METHOD PRIVATE REAL_TO_WHOLE_AND_FRACTION : BOOL
VAR_INPUT
	nReal		:	REAL;				// The real number you want to split into whole and fractional parts
END_VAR
VAR_OUTPUT
	nWhole		:	INT;				// The whole part of the input
	nFraction	:	UINT;				// The fractional part of the input (multiplied by 1000)
END_VAR
VAR
	sTemp		: STRING;
END_VAR
sTemp := REAL_TO_STRING(nReal);
nWhole := STRING_TO_INT(LEFT(sTEMP, FIND(sTemp, '.')));
sTemp := DELETE(sTEmp, FIND(sTemp, '.'), 1);
CASE LEN(sTemp) OF
	0:		sTemp := '000';
	1:		sTemp := CONCAT(sTemp, '00');
	2:		sTemp := CONCAT(sTemp, '0');
	ELSE	sTemp := LEFT(sTemp, 3);
END_CASE
nFraction := STRING_TO_UINT(sTemp);
REAL_TO_WHOLE_AND_FRACTION := TRUE;
END_METHOD

METHOD PRIVATE WHOLE_AND_FRACTION_TO_REAL : BOOL
VAR_INPUT
	nWhole		: INT;					// The whole part of the numbers you want to combine into real
	nFraction	: UINT;					// The fractional part of the numbers you want to combine into real
END_VAR
VAR_OUTPUT
	nReal 		: REAL;					// The result real number
END_VAR
VAR
	sTemp		: STRING;
END_VAR
nReal := STRING_TO_REAL(CONCAT(CONCAT(INT_TO_STRING(nWhole),'.'), UINT_TO_STRING(nFraction)));
WHOLE_AND_FRACTION_TO_REAL := TRUE;
END_METHOD

END_FUNCTION_BLOCK

// ---- POUs/CNC_1/CNC_1.TcPOU
PROGRAM CNC_1
VAR	(* Control *)
	nState						: UDINT;
	nStatePrevious				: UDINT;
	sState						: STRING(500);
	fbCycleTime					: TON;
	nCycleTime					: REAL;
	bError						: BOOL;
END_VAR
VAR (* LastStates *)
	anLastStates				: ARRAY[0..500] OF UDINT;
    iLastStates					: INT;
END_VAR
VAR (* Var IO *)
	{attribute 'TcLinkTo' := '		.fbMoveUpper.i_bBasePos	:= TIIB(13)^Channel 2^Input;
									.fbMoveUpper.i_bWorkPos	:= TIIB(13)^Channel 1^Input;
									.fbMoveUpper.q_bBasePos	:= TIIB(14)^Channel 2^Output;
									.fbMoveUpper.q_bWorkPos	:= TIIB(14)^Channel 1^Output;
									.fbMoveLower.i_bBasePos	:= TIIB(13)^Channel 4^Input;
									.fbMoveLower.i_bWorkPos	:= TIIB(13)^Channel 3^Input;
									.fbMoveLower.q_bBasePos	:= TIIB(14)^Channel 4^Output;
									.fbMoveLower.q_bWorkPos	:= TIIB(14)^Channel 3^Output;
									.fbLock.i_bBasePos	:= TIIB(13)^Channel 5^Input;
									.fbLock.i_bWorkPos	:= TIIB(13)^Channel 6^Input;
									.fbLock.q_bWorkPos	:= TIIB(14)^Channel 5^Output;
									.q_bToolCheckBlower := TIIB(14)^Channel 6^Output;
									.fbVisePos.arrRaw[0]	:= TIIB(10)^Module 1 (IOL_I_4byte)^TxPDO^input byte 0;	
									.fbVisePos.arrRaw[1] 	:= TIIB(10)^Module 1 (IOL_I_4byte)^TxPDO^input byte 1;
									.fbVisePos.arrRaw[2]	:= TIIB(10)^Module 1 (IOL_I_4byte)^TxPDO^input byte 2;
									.fbVisePos.arrRaw[3]	:= TIIB(10)^Module 1 (IOL_I_4byte)^TxPDO^input byte 3;
									.fbVisePos.nState		:= TIIB(10)^IO-Link DeviceState Inputs^Status of IO-Link Port 1;'}
	fbCncServoVise				: FB_CNC_Servo;	

END_VAR
VAR (* OPC_UA *)
	stCNC_Data					: POINTER TO OPC_CNC_Data_Collection;
	tHeartBeatDelay				: TON;
	bCNCHandshakeTimeout		:	BOOL;
	tCNCHandshakeTimer			:	TON;
	bCNCMidwareShutdownPossible	: 	BOOL;	//20, 40, 11400, 
	bShutdownIsProcessing		:	BOOL;
END_VAR
VAR	(*7 Axis Robot Communication*)
	bCNCRunning					:	BOOL;
END_VAR

(* OPC_UA *)
stCNC_Data := ADR(OPC_UA_CNC1);
tHeartBeatDelay(IN := stCNC_Data^.HeartBeat = 99, PT := T#500MS, Q=>);
IF tHeartBeatDelay.Q THEN
	stCNC_Data^.HeartBeat := 0;
END_IF

tCNCHandshakeTimer(		IN :=	(stCNC_Data^.HeartBeat = 0),
						PT := T#3S,
						Q=>bCNCHandshakeTimeout);
					
					
(* =================================== OPC_UA Automatic Shutdown handling =========================================== *)					
bCNCMidwareShutdownPossible := 	nState <= 10000;
								
IF bCNCMidwareShutdownPossible AND stCNC_Data^.MidwareRequestedShutdown AND (NOT bCNCHandshakeTimeout) THEN
	stCNC_Data^.ApproveShutdownRequest := TRUE;
END_IF

IF stCNC_Data^.ApproveShutdownRequest THEN
	IF bCNCHandshakeTimeout THEN
		bShutdownIsProcessing := TRUE;
	END_IF
END_IF

IF bShutdownIsProcessing THEN
	stCNC_Data^.ApproveShutdownRequest := FALSE;
	stCNC_Data^.MidwareRequestedShutdown := FALSE;
	IF (NOT bCNCHandshakeTimeout) THEN
		bShutdownIsProcessing := FALSE;
	END_IF
END_IF

(*Error handling*)
IF nState > 0 AND nState < 150000 THEN
	nStatePrevious := nState;
END_IF

(*Maintance*)
IF bManualMode THEN
	nState := 150000;
END_IF

(*Emergency*)
IF NOT i_bLO1_Main THEN
	nState := 0;
END_IF

(*Last states*)
IF(nState >= 1000) AND (nState < 150000) THEN
(*Steps before any state*)
	IF anLastStates[0] <> nState THEN
		FOR iLastStates:=500 TO 1 BY -1 DO
			anLastStates[iLastStates]:= anLastStates[iLastStates-1];
		END_FOR
		anLastStates[0]:= nState;
	END_IF
END_IF	

IF fbCncServoVise.bError (*OR stCNC_Data^.ControlStatus_Error*)
THEN
	bError  :=  TRUE;
END_IF

bCNCRunning := ((nState > 10000) AND (nState <= 30000));

CASE nState OF
{region "Alaphelyzet felvétel"}
	(****************************************************************************************)
	(******************************* Alaphelyzetfelvétel ************************************)
	(****************************************************************************************)	
	0:		(*-----=== Kimenetek törlése ===-----*)
		sState := CONCAT(UDINT_TO_STRING(nState) ,' - A biztonsági kör nem aktív');
		IF i_bLO1_Main AND NOT bManualMode THEN		//AND i_bLO1_CNC1 THEN		Nincs bekötve! Teszteléshez kikapcsolva! Ha a bekötés kész VISSZAÍRNI !!!!!!!!!!!!!!!
			stCNC_Data^.DoorControl_CloseDoor := FALSE;
			stCNC_Data^.DoorControl_OpenDoor := FALSE;
			stCNC_Data^.MagazineTable_Trigger := FALSE;
			stCNC_Data^.ToolTable_Trigger := FALSE;
			stCNC_Data^.M401_Acknowledge := FALSE;
			stCNC_Data^.M402_Acknowledge := FALSE;
			stCNC_Data^.M403_Acknowledge := FALSE;
			stCNC_Data^.StartCNCProgram := FALSE;
			stCNC_Data^.StopCNCProgram := FALSE;
			stCNC_Data^.CancelCNCProgram := FALSE;
			stCNC_Data^.SelectCNCProgramByNodeID := FALSE;
			stCNC_Data^.SelectCNCPrograBlockNumber := FALSE;
//			stCNC_Data^.ToolTablePath := '';
			stCNC_Data^.ToolTableLoadTrigger := FALSE;
			stCNC_Data^.MagazineTableLoadTrigger := FALSE;
			stCNC_Data^.ProgramLoadTrigger := FALSE;
			IF bStepEnable THEN
				nState := nState + 20;
			END_IF
		END_IF

	20:		(*-----=== CNC ellenőrzés ===-----*)
		sState := CONCAT(UDINT_TO_STRING(nState) ,' - A CNC ellenőrzése');
		IF stCNC_Data^.ServerState = 'Running' AND
		   stCNC_Data^.CurrentState_State = 'NCIsAvailable' THEN
				IF		stCNC_Data^.CurentState_Program = 'Running' THEN
					nState := 11500;										// A megmunkálás folyamatban -> Várakozás megmunkálás végére.
				ELSIF	stCNC_Data^.CurentState_Program = 'Idle' OR stCNC_Data^.CurentState_Program = 'NotSelected' OR stCNC_Data^.CurentState_Program = 'Interrupted' THEN
					IF (stDutData_Cnc1.nDutId > 0 AND stDutData_Cnc1.bDone) OR stDutData_Cnc1.bDutInVise THEN
						IF bStepEnable THEN									// Késztermék a satuban
							nState := 11560;
						END_IF
					ELSE
						IF bStepEnable THEN									// A satu üres
							nState := nState + 20;
						END_IF
					END_IF
				END_IF
		END_IF

	40:		(*-----=== CNC ajtó nnyitása ===-----*)
		sState := CONCAT(UDINT_TO_STRING(nState) ,' - A CNC ajtó nyitása');
		stCNC_Data^.DoorControl_OpenDoor := TRUE;
		IF stCNC_Data^.DoorControl_DoorOpened THEN
			IF bStepEnable THEN	
				stCNC_Data^.DoorControl_OpenDoor := FALSE;
				nState := nState + 20;
			END_IF
		END_IF

	60:
		nState := 10000;
{endregion}

{region "Alaphelyzet"}
	(****************************************************************************************)
	(*********************************** Alaphelyzet ****************************************)
	(****************************************************************************************)	
	10000:		(*-----=== Várakozás berakásra ===-----*)
		sState := CONCAT(UDINT_TO_STRING(nState) ,' - Várakozás alapanyagra');
		IF ((NOT bShutdownIsProcessing) AND (NOT stCNC_Data^.ApproveShutdownRequest)) THEN
			IF Robot7AxisProgram.bStartCNC1 THEN
				IF stDutData_Cnc1.nDutId > 0 THEN											// Alapanyag a robotnál
					IF bStepEnable THEN	
						nState := 11000;			// -> Alapanyag fogadása
					END_IF
				END_IF
			END_IF
		END_IF
{endregion}

{region "Alapanyag fogadása"}
	(****************************************************************************************)
	(******************************** Alapanyag fogadása ************************************)
	(****************************************************************************************)	
	11000:		(*-----=== Satu pozícionálása ===-----*)
		sState := CONCAT(UDINT_TO_STRING(nState) ,' - Satu pozícionálása');
		fbCncServoVise.nPosition := stDutData_Cnc1.nDimX;
		fbCncServoVise.eCommand := E_CncServoCommand.MovePos;
		IF fbCncServoVise.bDone THEN
			IF bStepEnable THEN
				fbCncServoVise.eCommand := E_CncServoCommand.NoCommand;
				nState := 11100;
			END_IF
		END_IF

	11100:		(*-----=== Várakozás alapanyag berakásra ===-----*)
		sState := CONCAT(UDINT_TO_STRING(nState) ,' - Alapanyag berakás');
		IF Robot7AxisProgram.fbRobot.bZoneCnc1 THEN
			IF bStepEnable THEN
				stDutData_Cnc1.bDutInVise := TRUE;
				nState := 11200;
			END_IF
		END_IF

	11200:		(*-----=== Várakozás robot távozásra ===-----*)
		sState := CONCAT(UDINT_TO_STRING(nState) ,' - Várakozás robot távozásra');
		IF NOT Robot7AxisProgram.fbRobot.bZoneCnc1 THEN
			IF bStepEnable THEN
				nState := 11300;
			END_IF
		END_IF
	
	11300:		(*-----=== Satu rögzítése ===-----*)
		sState := CONCAT(UDINT_TO_STRING(nState) ,' - Satu rögzítése');
		fbCncServoVise.nTorque := stDutData_Cnc1.nTorque;
		fbCncServoVise.eCommand := E_CncServoCommand.Fixed;
		IF fbCncServoVise.bDone THEN
			IF bStepEnable THEN
				fbCncServoVise.eCommand := E_CncServoCommand.NoCommand;
				nState := 11400;
			END_IF
		END_IF

	11400:		(*-----=== CNC ajtó zárása ===-----*)
		sState := CONCAT(UDINT_TO_STRING(nState) ,' - A CNC ajtó zárása');
		stCNC_Data^.DoorControl_CloseDoor := TRUE;
		IF stCNC_Data^.DoorControl_DoorClosed THEN
			IF bStepEnable THEN	
				stCNC_Data^.DoorControl_CloseDoor := FALSE;
				nState := nState + 20;
			END_IF
		END_IF

	11420:		(*-----=== CNC előkészítése ===-----*)
		sState := CONCAT(UDINT_TO_STRING(nState) ,' - A CNC előkészítése');
		IF TRUE THEN															// Külön FB-be rakni mert még képlékeny CAM file letöltése, ellenőrzése, felmásolása, betöltése, ........ 
			IF bStepEnable THEN	
				nState := nState + 20;
			END_IF
		END_IF

	11440:		(*-----=== CAM program indítása ===-----*)
		sState := CONCAT(UDINT_TO_STRING(nState) ,' - CAM program indítása');
		stCNC_Data^.StartCNCProgram := TRUE;
		IF stCNC_Data^.CurentState_Program = 'Running' THEN
			IF bStepEnable THEN	
				stCNC_Data^.StartCNCProgram := FALSE;
				nState := 11500;
			END_IF
		END_IF
	
	11500:		(*-----=== Várakozás CAM program végére ===-----*)
		sState := CONCAT(UDINT_TO_STRING(nState) ,' - Várakozás CAM program végére');
		IF stCNC_Data^.CurentState_Program = 'Finished' OR stCNC_Data^.CurentState_Program = 'Idle' THEN
			IF bStepEnable THEN	
				stCNC_Data^.DoorControl_CloseDoor := FALSE;
				nState := nState + 20;
			END_IF
		END_IF

	11520:		(*-----=== CNC folyamat befejezése ===-----*)
		sState := CONCAT(UDINT_TO_STRING(nState) ,' - A CNC folyamat befejezése');
		IF TRUE THEN															// Külön FB-be rakni mert még képlékeny: minőségellenőrzés, mérési adatok, .... 
			IF bStepEnable THEN	
				nState := nState + 20;
			END_IF
		END_IF

	11540:		(*-----=== CAM program leállítása ===-----*)
		sState := CONCAT(UDINT_TO_STRING(nState) ,' - CAM program leállítása');
		stCNC_Data^.CancelCNCProgram := TRUE;
		IF stCNC_Data^.CurentState_Program = 'Idle' THEN
			IF bStepEnable THEN	
				stCNC_Data^.CancelCNCProgram := FALSE;
				nState := nState + 20;
			END_IF
		END_IF

	11560:		(*-----=== CNC ajtó nnyitása ===-----*)
		sState := CONCAT(UDINT_TO_STRING(nState) ,' - A CNC ajtó nyitása');
		stCNC_Data^.DoorControl_OpenDoor := TRUE;
		IF stCNC_Data^.DoorControl_DoorOpened THEN
			IF bStepEnable THEN	
				stCNC_Data^.DoorControl_OpenDoor := FALSE;
				nState := 11600;
			END_IF
		END_IF
	
	11600:		(*-----=== Satu pozícionálása ===-----*)
		sState := CONCAT(UDINT_TO_STRING(nState) ,' - Satu pozícionálása');
		fbCncServoVise.nPosition := stDutData_Cnc1.nDimX;
		fbCncServoVise.eCommand := E_CncServoCommand.MovePos;
		IF fbCncServoVise.bDone THEN
			IF bStepEnable THEN
				stDutData_Cnc1.bDone := TRUE;
				stDutData_Cnc1.bPass := TRUE;
				fbCncServoVise.eCommand := E_CncServoCommand.NoCommand;
				nState := 12000;
			END_IF
		END_IF
{endregion}

{region "Alapanyag küldése"}
	(****************************************************************************************)
	(******************************** Alapanyag küldése ************************************)
	(****************************************************************************************)	
	12000:		(*-----=== Várakozás alapanyag kivételre ===-----*)
		sState := CONCAT(UDINT_TO_STRING(nState) ,' - Alapanyag kivétel');
		IF Robot7AxisProgram.fbRobot.bZoneCnc1 THEN
			IF bStepEnable THEN
				nState := 12100;
			END_IF
		END_IF
	
	12100:		(*-----=== Várakozás robot távozásra ===-----*)
		sState := CONCAT(UDINT_TO_STRING(nState) ,' - Satu rögzítése');
		IF NOT Robot7AxisProgram.fbRobot.bZoneCnc1 THEN
			IF bStepEnable THEN
				stDutData_Cnc1.bDutInVise := FALSE;
				stDutData_Cnc1.nDutId := 0;
				stDutData_Cnc1.bDone := FALSE;
				nState := 10000;
			END_IF
		END_IF
{endregion}

	150000: (* Maintenance *)
		sState := CONCAT(UDINT_TO_STRING(nState) ,' - Maintenance');
		IF NOT bManualMode THEN
			nState := 0;
		END_IF
		
	200000:(* Error handling *)
		sState := CONCAT(UDINT_TO_STRING(nState) ,CONCAT(' - Error, from this state: ' , sState));
		nState := 200020;

	200020:(* Error handling *)
		IF bAckP THEN
			CASE nStatePrevious OF
				0..9999: nState := 0;
//				10000..25000: nState := 10000;
//				30000..31000: nState := 30000;
			ELSE nState := 0;
			END_CASE
		END_IF	
		
	ELSE //Not a real step, for test purposes
		sState := CONCAT(UDINT_TO_STRING(nState) ,' - Not a real step, for test purposes');
END_CASE

(*Timers***************************************************)
fbCycleTime(IN:= nState > 10000 AND nState <= 95000, PT:= T#1D, Q=> , ET=> );
IF nState > 10000 AND nState <= 95000 THEN
	nCycleTime := TIME_TO_REAL(fbCycleTime.ET)/1000;
END_IF

ServoVise();
//fbCncServoVise.bTestUp := i_bTest_Up;
//fbCncServoVise.bTestDown := i_bTest_Down;
//fbCncServoVise.bTestStop := i_bTest_Stop;

ACTION ServoVise:
fbCncServoVise(
	sName:= 'AWEA_1', 
	bErrorAck:= bAckP, 
	bEnable:= i_bLO1_Main,		//AND i_bLO1_CNC1 THEN		Nincs bekötve! Teszteléshez kikapcsolva! Ha a bekötés kész VISSZAÍRNI !!!!!!!!!!!!!!!, 
	bManualMode:= bManualMode, 
	bReady=> , 
	bBusy=> , 
	bDone=> , 
	bError=> );
END_ACTION

END_PROGRAM

// ---- POUs/FBs/CNC_Servo/FB_CNC_Servo.TcPOU
FUNCTION_BLOCK FB_CNC_Servo
VAR_INPUT
	sName						: STRING;
	eCommand					: E_CncServoCommand;
	nPosition					: LREAL;				// Termék nominális mérete
	nTorque						: REAL;					// Meghúzási nyomaték
	bErrorAck					: BOOL;
	bEnable						: BOOL;
	bManualMode					: BOOL;
	nCalOffset_1				: LREAL := 22.32;
	nCalOffset_2				: LREAL := 99.01;
END_VAR
VAR	(* Control *)
	nState						:UDINT;
	nStatePrevious				:UDINT;
	sState						:STRING(500);
	fbCycleTime					:TON;
	nCycleTime					:REAL;
END_VAR
VAR //LastStates
	anLastStates				:ARRAY[0..500] OF UDINT;
    iLastStates					:INT;
END_VAR
VAR_OUTPUT
	bReady						: BOOL;
	bBusy 						: BOOL;
	bDone 						: BOOL;
	bError 						: BOOL;
END_VAR
VAR
	fbMoveUpper					: FB_Bistabil;
	fbMoveLower					: FB_Bistabil;
	fbLock						: FB_Bistabil;
	fbVisePos					: FB_BTL1AR0;
	fbServoVise					: FB_ServoVise;
	q_bToolCheckBlower 	AT %Q*	: BOOL;		// Szerszám ellenőrző tisztítás
	bRotate						: BOOL := FALSE;
	tAttach						: TON;
	tFillUp						: TON;
END_VAR

(* Timers *)
tAttach(IN:= fbMoveLower.bWorkPosCmd AND fbMoveUpper.bWorkPosCmd AND NOT bRotate, PT:= T#5000MS, Q=> , ET=> );
tFillUp(IN:= fbMoveLower.bWorkPosCmd AND fbMoveLower.bBasePosCmd, PT:= T#800MS, Q=> , ET=> );

(*CNC Servo Offset Adjustment*)
fbServoVise.nCalOffset_1 := nCalOffset_1;
fbServoVise.nCalOffset_2 := nCalOffset_2;

(*Error handling*)
IF nState > 0 AND nState < 150000 THEN
	nStatePrevious := nState;
END_IF

(*Maintance*)
IF bManualMode THEN
	nState := 150000;
END_IF

(*Emergency*)
IF NOT bEnable THEN
	nState := 0;
END_IF

(*Last states*)
IF(nState >= 1000) AND (nState < 150000) THEN
(*Steps before any state*)
	IF anLastStates[0] <> nState THEN
		FOR iLastStates:=500 TO 1 BY -1 DO
			anLastStates[iLastStates]:= anLastStates[iLastStates-1];
		END_FOR
		anLastStates[0]:= nState;
	END_IF
END_IF	

IF fbMoveUpper.bError OR fbMoveLower.bError OR fbLock.bError OR fbServoVise.bError
THEN
	bError  :=  TRUE;
END_IF



CASE nState OF
{region "Alaphelyzet felvétel"}
	(****************************************************************************************)
	(******************************* Alaphelyzetfelvétel ************************************)
	(****************************************************************************************)	
	0:		(*-----=== Kimenetek törlése ===-----*)
		sState := CONCAT(UDINT_TO_STRING(nState) ,' - A biztonsági kör nem aktív');
		bReady := FALSE;
		bBusy := FALSE;
		bDone := FALSE;
		fbLock.bBasePosCmd := FALSE;
		fbLock.bWorkPosCmd := FALSE;
		fbMoveLower.bBasePosCmd := FALSE;
		fbMoveLower.bWorkPosCmd := FALSE;
		fbMoveUpper.bBasePosCmd := FALSE;
		fbMoveUpper.bWorkPosCmd := FALSE;
		fbServoVise.eCommand := E_ServoVise_Command.NoCommand;
		IF bEnable THEN
			IF bStepEnable THEN
				nState := nState + 20;
			END_IF
		END_IF

	20:		(*-----=== Alaphelyzet ellenőrzés ===-----*)
		sState := CONCAT(UDINT_TO_STRING(nState) ,' - Alaphelyzetfelvétel: - Hengerek ellenőrzése');
		IF	fbLock.i_bBasePos AND
			fbMoveLower.i_bBasePos AND
			fbMoveUpper.i_bBasePos THEN
					fbLock.bBasePosCmd := TRUE;									// Hengerek alaphelyzetben -> Vezérlést ráadni és hajrá!!
					fbLock.bWorkPosCmd := FALSE;
					fbMoveLower.bBasePosCmd := TRUE;
					fbMoveLower.bWorkPosCmd := FALSE;
					fbMoveUpper.bBasePosCmd := TRUE;
					fbMoveUpper.bWorkPosCmd := FALSE;
					IF bStepEnable THEN
						nState := 60;
					END_IF
		ELSIF	fbMoveLower.i_bBasePos AND
				fbMoveUpper.i_bBasePos THEN
					fbLock.bBasePosCmd := FALSE;								// Hengerek munkahelyzetben -> Vezérlést ráadni és hajrá!! 
					fbLock.bWorkPosCmd := TRUE;
					fbMoveLower.bBasePosCmd := FALSE;
					fbMoveLower.bWorkPosCmd := TRUE;
					fbMoveUpper.bBasePosCmd := FALSE;
					fbMoveUpper.bWorkPosCmd := TRUE;
					IF bStepEnable THEN
						nState := nState + 40;
					END_IF
		ELSE
					fbLock.bBasePosCmd := FALSE;								// Hengerek se itt se ott -> feltöltés szükséges
					fbLock.bWorkPosCmd := TRUE;
					fbMoveLower.bBasePosCmd := TRUE;
					fbMoveLower.bWorkPosCmd := TRUE;
					fbMoveUpper.bBasePosCmd := TRUE;
					fbMoveUpper.bWorkPosCmd := TRUE;
					IF bStepEnable THEN
						nState := nState + 20;
					END_IF
		END_IF
	
	40:		(*-----=== Hengerek feltöltése ===-----*)
		sState := CONCAT(UDINT_TO_STRING(nState) ,' - Alaphelyzetfelvétel: - Hengerek feltöltése');
		IF tFillUp.Q THEN
			fbMoveLower.bBasePosCmd := TRUE;
			fbMoveLower.bWorkPosCmd := FALSE;
			fbMoveUpper.bBasePosCmd := TRUE;
			fbMoveUpper.bWorkPosCmd := FALSE;
			nState := nState + 20;
		END_IF

	
	60:		(*-----=== fbLock munkahelyzetbe ===-----*)
		sState := CONCAT(UDINT_TO_STRING(nState) ,' - Alaphelyzetfelvétel: - Lock henger munkahelyzetbe');
		fbLock.bBasePosCmd := FALSE;
		fbLock.bWorkPosCmd := TRUE;
		IF fbLock.bWorkPosStab THEN
			IF bStepEnable THEN
				nState := nState + 20;
			END_IF
		END_IF
		
	80:		(*-----=== fbMoveLower & fbMoveUpper alaphelyzetbe ===-----*)
		sState := CONCAT(UDINT_TO_STRING(nState) ,' - Alaphelyzetfelvétel: - Mozgató hengerek alaphelyzetbe');
		fbMoveLower.bBasePosCmd := TRUE;
		fbMoveLower.bWorkPosCmd := FALSE;
		fbMoveUpper.bBasePosCmd := TRUE;
		fbMoveUpper.bWorkPosCmd := FALSE;
		IF fbMoveLower.bBasePosStab AND fbMoveUpper.bBasePosStab THEN
			IF bStepEnable THEN
				nState := nState + 20;
			END_IF
		END_IF

	100:		(*-----=== fbLock alaphelyzetbe ===-----*)
		sState := CONCAT(UDINT_TO_STRING(nState) ,' - Alaphelyzetfelvétel: - Lock henger alaphelyzetbe');
		fbLock.bBasePosCmd := TRUE;
		fbLock.bWorkPosCmd := FALSE;
		IF fbLock.bBasePosStab THEN
			IF bStepEnable THEN
				bBusy := FALSE;
				bDone := TRUE;
				nState := 10000;
			END_IF
		END_IF
{endregion}

{region "Alaphelyzet"}
	(****************************************************************************************)
	(*********************************** Alaphelyzet ****************************************)
	(****************************************************************************************)	
	10000:		(*-----=== Várakozás parancsra ===-----*)
		sState := CONCAT(UDINT_TO_STRING(nState) ,' - Alaphelyzet, várakozás parancsra');
		IF eCommand = E_CncServoCommand.NoCommand THEN
				bReady := TRUE;
				bBusy := FALSE;
				bDone := FALSE;
		ELSIF eCommand = E_CncServoCommand.Base THEN
				bBusy := TRUE;
				nState := 11000;
		ELSE
				bBusy := TRUE;
				nState := 12000;
		END_IF
		
{endregion}

{region "Alaphelyzetbe mozgás"}
	(****************************************************************************************)
	(***************************** Alaphelyzetbe mozgás *************************************)
	(****************************************************************************************)	
	11000:		(*-----=== fbLock munkahelyzetbe ===-----*)
		sState := CONCAT(UDINT_TO_STRING(nState) ,' - Lock henger munkahelyzetbe');
		fbLock.bBasePosCmd := FALSE;
		fbLock.bWorkPosCmd := TRUE;
		IF fbLock.bWorkPosStab THEN
			IF bStepEnable THEN
				nState := nState + 20;
			END_IF
		END_IF
		
	11020:		(*-----=== fbMoveLower & fbMoveUpper alaphelyzetbe ===-----*)
		sState := CONCAT(UDINT_TO_STRING(nState) ,' - Mozgató hengerek alaphelyzetbe');
		fbMoveLower.bBasePosCmd := TRUE;
		fbMoveLower.bWorkPosCmd := FALSE;
		fbMoveUpper.bBasePosCmd := TRUE;
		fbMoveUpper.bWorkPosCmd := FALSE;
		IF fbMoveLower.bBasePosStab AND fbMoveUpper.bBasePosStab THEN
			IF bStepEnable THEN
				nState := nState + 20;
			END_IF
		END_IF

	11040:		(*-----=== fbLock alaphelyzetbe ===-----*)
		sState := CONCAT(UDINT_TO_STRING(nState) ,' - Lock henger alaphelyzetbe');
		fbLock.bBasePosCmd := TRUE;
		fbLock.bWorkPosCmd := FALSE;
		IF fbLock.bBasePosStab THEN
			IF bStepEnable THEN
				bBusy := FALSE;
				bDone := TRUE;
				nState := nState + 20;
			END_IF
		END_IF
	
	11060:		(*-----=== Várakozás parancstörlésre ===-----*)
		sState := CONCAT(UDINT_TO_STRING(nState) ,' - Várakozás parancs törlésre');
		IF eCommand = E_CncServoCommand.NoCommand THEN
			bBusy := FALSE;
			bDone := FALSE;
			nState := 10000;
		END_IF
{endregion}

{region "Satu Csatlakoztatás"}
	(****************************************************************************************)
	(***************************** Satu Csatlakoztatás **************************************)
	(****************************************************************************************)	
	12000:		(*-----=== Csatlakoztatás ellenőrzése ===-----*)
		sState := CONCAT(UDINT_TO_STRING(nState) ,' - Csatlakoztatás ellenőrzése');
		IF fbMoveLower.bWorkPosStab AND fbMoveUpper.bWorkPosStab THEN
			IF bStepEnable THEN
				nState := 12200;							// A szervo már csatlakoztatva van
			END_IF
		ELSE
			IF bStepEnable THEN
				IF bRotate THEN
					nState := nState + 20;					// A szervó alaphelyzetbe van -> csatlakoztatás forgatással
				ELSE
					nState := nState + 40;					// A szervó alaphelyzetbe van -> csatlakoztatás forgatás nélkül
				END_IF
			END_IF
		END_IF

	12020:		(*-----=== fbServoVise csatlakoztatás program indítása ===-----*)
		sState := CONCAT(UDINT_TO_STRING(nState) ,' - Csatlakoztatási segédmozgás indítása');
		fbServoVise.eCommand := E_ServoVise_Command.Attach;
		IF fbServoVise.bDone THEN
			IF bStepEnable THEN
				nState := nState + 20;
			END_IF
		END_IF

	12040:		(*-----=== fbLock munkahelyzetbe ===-----*)
		sState := CONCAT(UDINT_TO_STRING(nState) ,' - Lock henger munkahelyzetbe');
		fbLock.bBasePosCmd := FALSE;
		fbLock.bWorkPosCmd := TRUE;
		IF fbLock.bWorkPosStab THEN
			IF bStepEnable THEN
				nState := nState + 20;
			END_IF
		END_IF
		
	12060:		(*-----=== fbMoveLower & fbMoveUpper munkahelyzetbe ===-----*)
		sState := CONCAT(UDINT_TO_STRING(nState) ,' - Mozgató hengerek munkahelyzetbe');
		fbMoveLower.bBasePosCmd := FALSE;
		fbMoveLower.bWorkPosCmd := TRUE;
		fbMoveUpper.bBasePosCmd := FALSE;
		fbMoveUpper.bWorkPosCmd := TRUE;
		IF fbMoveLower.bWorkPosStab AND fbMoveUpper.bWorkPosStab THEN
			IF bStepEnable THEN
				nState := nState + 20;
			END_IF
		ELSIF tAttach.Q THEN										// Sikertelen csatlakozás -> Szervo bekapcsolása
			IF bStepEnable THEN
				bRotate := TRUE;
				nState := 12000;
			END_IF
		END_IF

	12080:		(*-----=== fbServoVise csatlakoztatás program leállítása ===-----*)
		sState := CONCAT(UDINT_TO_STRING(nState) ,' - Csatlakoztatási segédmozgás leállítása');
		fbServoVise.eCommand := E_ServoVise_Command.NoCommand;
		IF NOT fbServoVise.bDone THEN
			IF bStepEnable THEN
				bRotate := FALSE;
				nState := 12200;
			END_IF
		END_IF

	12200:		(*-----=== A parancs ellenőrzése ===-----*)
		IF fbVisePos.bValid THEN								// Csak ha az útmérő is észhez tért!  Egy timeout kell majd mert hátha egyszer megdöglik!!!!!
			IF eCommand = E_CncServoCommand.NoCommand THEN
					nState := 10000;
			ELSIF eCommand = E_CncServoCommand.Base THEN
					nState := 11000;
			ELSIF eCommand = E_CncServoCommand.MovePos THEN
					nState := 13000;
			ELSIF eCommand = E_CncServoCommand.Fixed THEN
					nState := 14000;
			ELSIF eCommand = E_CncServoCommand.Release THEN
					nState := 15000;
			END_IF
		END_IF
{endregion}

{region "Satu pozícionálás"}
	(****************************************************************************************)
	(******************************** Satu pozícionálás *************************************)
	(****************************************************************************************)	
	13000:		(*-----=== Pozícionálás indítása ===-----*)
		sState := CONCAT(UDINT_TO_STRING(nState) ,' - Satu pozícionálása');
		fbServoVise.eCommand := E_ServoVise_Command.MoveToPos;
		IF fbServoVise.bDone THEN
			IF bStepEnable THEN
				fbServoVise.eCommand := E_ServoVise_Command.NoCommand;
				bRotate := FALSE;
				nState := 11000;
			END_IF
		END_IF
{endregion}

{region "Satu Rögzytés"}
	(****************************************************************************************)
	(*********************************** Satu Rögzítés **************************************)
	(****************************************************************************************)	
	14000:		(*-----=== Rögzítés indítása ===-----*)
		sState := CONCAT(UDINT_TO_STRING(nState) ,' - Satu rögzítése');
		fbServoVise.eCommand := E_ServoVise_Command.Fix;
		IF fbServoVise.bDone THEN
			IF bStepEnable THEN
				fbServoVise.eCommand := E_ServoVise_Command.NoCommand;
				bRotate := FALSE;
				nState := 11000;
			END_IF
		END_IF
{endregion}

{region "Satu Kioldás"}
	(****************************************************************************************)
	(************************************ Satu Kioldás **************************************)
	(****************************************************************************************)	
	15000:		(*-----=== Kioldás indítása ===-----*)
		sState := CONCAT(UDINT_TO_STRING(nState) ,' - Satu kioldása');
		fbServoVise.eCommand := E_ServoVise_Command.Release;
		IF fbServoVise.bDone THEN
			IF bStepEnable THEN
				fbServoVise.eCommand := E_ServoVise_Command.NoCommand;
				bRotate := FALSE;
				nState := 11000;
			END_IF
		END_IF
{endregion}

	150000: (* Maintenance *)
		sState := CONCAT(UDINT_TO_STRING(nState) ,' - Maintenance');
		IF NOT bManualMode THEN
			nState := 0;
		END_IF
		
	200000:(* Error handling *)
		sState := CONCAT(UDINT_TO_STRING(nState) ,CONCAT(' - Error, from this state: ' , sState));
		nState := 200020;

	200020:(* Error handling *)
		IF bAckP THEN
			CASE nStatePrevious OF
				0..9999: nState := 0;
//				10000..25000: nState := 10000;
//				30000..31000: nState := 30000;
			ELSE nState := 0;
			END_CASE
		END_IF	
		
	ELSE //Not a real step, for test purposes
		sState := CONCAT(UDINT_TO_STRING(nState) ,' - Not a real step, for test purposes');
END_CASE

Servo();
Pneu();

ACTION Pneu:
fbMoveUpper(
	sName:= , 
	sBasePosSensor:= , 
	sWorkPosSensor:= , 
	bEn:= bEnable, 
	bEHA:= NOT bManualMode AND NOT fbMoveUpper.bWorkPosCmd, 
	nEHMode:= , 
	bDisableManualCmd:= NOT bManualMode, 
	bBasePosCmd:= , 
	bWorkPosCmd:= , 
	bAck:= bErrorAck, 
	timBasePos:= , 
	timWorkPos:= , 
	timBasePosStab:= , 
	timWorkPosStab:= , 
	i_bBasePos:= , 
	i_bWorkPos:= , 
	sSourceName:= , 
	stBasePosEvent:= , 
	stWorkPosEvent:= , 
	bBasePosStab=> , 
	bWorkPosStab=> , 
	bError=> , 
	sError=> , 
	q_bBasePos=> , 
	q_bWorkPos=> );

fbMoveLower(
	sName:= , 
	sBasePosSensor:= , 
	sWorkPosSensor:= , 
	bEn:= bEnable, 
	bEHA:= NOT bManualMode AND NOT fbMoveLower.bWorkPosCmd, 
	nEHMode:= , 
	bDisableManualCmd:= NOT bManualMode, 
	bBasePosCmd:= , 
	bWorkPosCmd:= , 
	bAck:= bErrorAck, 
	timBasePos:= , 
	timWorkPos:= , 
	timBasePosStab:= , 
	timWorkPosStab:= , 
	i_bBasePos:= , 
	i_bWorkPos:= , 
	sSourceName:= , 
	stBasePosEvent:= , 
	stWorkPosEvent:= , 
	bBasePosStab=> , 
	bWorkPosStab=> , 
	bError=> , 
	sError=> , 
	q_bBasePos=> , 
	q_bWorkPos=> );

fbLock(
	sName:= , 
	sBasePosSensor:= , 
	sWorkPosSensor:= , 
	bEn:= bEnable, 
	bEHA:= NOT bManualMode, 
	nEHMode:= , 
	bDisableManualCmd:= NOT bManualMode, 
	bBasePosCmd:= , 
	bWorkPosCmd:= , 
	bAck:= bErrorAck, 
	timBasePos:= , 
	timWorkPos:= , 
	timBasePosStab:= , 
	timWorkPosStab:= , 
	i_bBasePos:= , 
	i_bWorkPos:= , 
	sSourceName:= , 
	stBasePosEvent:= , 
	stWorkPosEvent:= , 
	bBasePosStab=> , 
	bWorkPosStab=> , 
	bError=> , 
	sError=> , 
	q_bBasePos=> , 
	q_bWorkPos=> );
END_ACTION

ACTION Servo:
fbVisePos();
fbServoVise(
	bErrorAck:= bAckP, 
	bEnable:= bEnable, 
	eCommand:= , 
	bManualMode:= bManualMode, 
	lrTargetDistance:= nPosition, 
	lrVisePosition:= fbVisePos.nDistance, 
	bVisePosValid:= fbVisePos.bValid, 
	nTargetVelocity:= 4, 
	nTorque:= nTorque, 
	nTorqueRamp:= 10, 
	nTorqueVelocityLimit:= 0.5, 
	nOverride:= 100, 
	nAttachVelocity:= 0.05, 
	stAxisEvent:= , 
	bReady=> , 
	bBusy=> , 
	bDone=> , 
	bError=> );
END_ACTION

END_FUNCTION_BLOCK

// ---- POUs/FBs/Pneumatics/FB_Bistabil.TcPOU
FUNCTION_BLOCK FB_Bistabil
VAR_INPUT
	sName				:STRING(50);
	sBasePosSensor		:STRING(10);		(*Base position sensor*)
	sWorkPosSensor		:STRING(10);		(*Work position sensor*)
	bEn					:BOOL;				(*Enable signal*)
	bEHA				:BOOL; 				(*Error-handling active *)
	nEHMode				:BYTE;				(*0: Delete output commant, 1: Control device to the opposite direction, 2: No change control if an error occurs*)
	bDisableManualCmd	:BOOL;				(*Manual control disable*)
	bBasePosCmd			:BOOL;				(*Control to Base pos*)
	bWorkPosCmd			:BOOL;				(*Control to work pos*)
	bAck				:BOOL; 				(*Acknowledge*)
	timBasePos			:TIME:=T#5S;		(*Time for base position*)
	timWorkPos			:TIME:=T#5S;		(*Time fort work position*)
	timBasePosStab		:TIME:=T#200MS;		(*Time to set base position*)
	timWorkPosStab		:TIME:=T#200MS;		(*Time to set work position*)
	i_bBasePos			AT %I*	:BOOL;		(*Base position*)
	i_bWorkPos			AT %I*	:BOOL;		(*Work position*)
	sSourceName			:STRING(10);		(*Station name - if there are multiple monitors*)
	stBasePosEvent		:TcEventEntry;		(*Event definition*)
	stWorkPosEvent		:TcEventEntry;		(*Event definition*)
END_VAR
VAR_OUTPUT
	bBasePosStab		:BOOL;				(*Base position stabil*)
	bWorkPosStab		:BOOL;				(*Work position stabil*)
	bError				:BOOL;				(*Error*)
	sError				:STRING(255);		(*Error string*)
	q_bBasePos			AT %Q*	:BOOL;		(*Control to base position*)
	q_bWorkPos			AT %Q*	:BOOL;		(*Control to work position*)
END_VAR
VAR
	tBP, tWP, tDPWP		:TON;
	tBPS, tWPS			:TON;
	bErrBasePos0		:BOOL;				(*Base position error 0: the signal did not stop after reaching base position*)
	bErrBasePos1		:BOOL;				(*Base position error 1: the signal did not appear while reaching base position*)
	bErrWorkPos0		:BOOL; 				(*Work position error 0: the signal did not stop after reaching work position*)
	bErrWorkPos1		:BOOL; 				(*Work position error 1: the signal did not appear while reaching work position*)
	bErrBPWP			:BOOL;				(*To positions at the same time error*)
	bIsInitalized		:BOOL;
	fbBasePosAlarm		:FB_TcAlarm;
	fbWorkPosAlarm		:FB_TcAlarm;
	fbSource			:FB_TcSourceInfo;
END_VAR

(*	Documentation
	--------------------------------------------------------------------------------
	Info		:	FB cylinders, bistabil, monostabil 
	Name		:	FB_Bistabil
	Modifier	:	Gyarmati Péter
	Date		:	2022.06.20
	Revision	:	1.32
	--------------------------------------------------------------------------------
	Requirements:	-
	Variable	:	-
	Visu		:	-
	UserControl	:	-
	--------------------------------------------------------------------------------
	Details		:	Alarms included. 
					Strings modified, to reduce the size of the FB.
					The error handling was modified because of the language change (only base and work position errors set)
					sSourceName -> It adds the stations name to the string after an error. 
	--------------------------------------------------------------------------------
	Usage		:	For example.:
					fbPaletteLift(
						sName:= 'Palette lifter', 
						bEn:= bEmyOK, 
						bEHA:= bGlobalEHA, 
						bDisableManualCmd:= NOT bManualMode, 
						bAck:= bAckP,  
						stBasePosEvent:= TC_Events.MyEvents.Valve_1,
						stWorkPosEvent:= TC_Events.MyEvents.Valve_2);
*)

(*Error handling Tc3_EventLogger*)
IF NOT bIsInitalized THEN
	bIsInitalized := TRUE;
	fbSource.sName := sSourceName;
	IF sSourceName = '' THEN
		fbBasePosAlarm.CreateEx(stBasePosEvent, TRUE, 0);
		fbWorkPosAlarm.CreateEx(stWorkPosEvent, TRUE, 0);
	ELSE
		fbBasePosAlarm.CreateEx(stBasePosEvent, TRUE, fbSource);
		fbWorkPosAlarm.CreateEx(stWorkPosEvent, TRUE, fbSource);		
		// This Addstring part puts the SourceName in a bracket. This is only required if there are multiple stations/monitort and this is how they are separated.
		fbBasePosAlarm.ipArguments.Clear().AddString(sSourceName);
		fbWorkPosAlarm.ipArguments.Clear().AddString(sSourceName);		
	END_IF
END_IF

(*Error acknowledge*)
IF bAck OR NOT bEHA THEN
	bErrBasePos0 := FALSE;
	bErrWorkPos0 := FALSE;
	bErrBasePos1 := FALSE;
	bErrWorkPos1 := FALSE;
	bErrBPWP := FALSE;
	IF fbBasePosAlarm.eConfirmationState = 2 THEN
		fbBasePosAlarm.Confirm(0);
	END_IF	
	IF fbWorkPosAlarm.eConfirmationState = 2 THEN
		fbWorkPosAlarm.Confirm(0);
	END_IF
END_IF

(*Error setting base position*)
tBP(IN:= bEn AND bEHA AND q_bBasePos AND NOT q_bWorkPos, PT:= timBasePos);

IF tBP.Q AND NOT i_bBasePos THEN
	bErrBasePos1 := TRUE;
	IF (fbBasePosAlarm.eConfirmationState <> 2 AND fbBasePosAlarm.nTimeCleared <> 0 AND fbBasePosAlarm.nTimeConfirmed <> 0) OR //Ha már volt alarm, akkor van bennük érték
		(fbBasePosAlarm.eConfirmationState = 1 AND fbBasePosAlarm.nTimeCleared = 0 AND fbBasePosAlarm.nTimeConfirmed = 0)	//Első futás esetén
	THEN
		fbBasePosAlarm.Raise(0);
	END_IF
END_IF

IF tBP.Q AND i_bWorkPos THEN
	//bErrWorkPos0 := TRUE;
END_IF

(*Error setting work position*)
tWP(IN:= bEn AND bEHA AND q_bWorkPos AND NOT q_bBasePos , PT:= timWorkPos);

IF tWP.Q AND NOT i_bWorkPos THEN
	bErrWorkPos1 := TRUE;
	IF (fbWorkPosAlarm.eConfirmationState <> 2 AND fbWorkPosAlarm.nTimeCleared <> 0 AND fbWorkPosAlarm.nTimeConfirmed <> 0) OR //Ha már volt alarm, akkor van bennük érték
		(fbWorkPosAlarm.eConfirmationState = 1 AND fbWorkPosAlarm.nTimeCleared = 0 AND fbWorkPosAlarm.nTimeConfirmed = 0)	//Első futás esetén
	THEN
		fbWorkPosAlarm.Raise(0);
	END_IF
END_IF

IF tWP.Q AND i_bBasePos THEN
	//bErrBasePos0 := TRUE;
END_IF

(*Two work positions at the same time*)
tDPWP(In:= bEn AND bEHA AND i_bBasePos AND i_bWorkPos, PT:= T#600MS);

IF tDPWP.q THEN
	//bErrBPWP := TRUE;
END_IF;

bError := bErrBasePos0 OR bErrWorkPos0 
	OR bErrBasePos1 OR bErrWorkPos1
	OR bErrBPWP;

(*Control*)
CASE nEHMode OF
	0:	(*Cancels control if an error occurs*)
		IF bEn AND bBaseposCmd AND (NOT bEHA OR NOT bError) THEN
			q_bBasePos := TRUE;
		ELSE
			q_bBasePos := FALSE;
		END_IF
		IF bEn  AND bWorkPosCmd AND (NOT bEHA OR NOT bError) THEN
			q_bWorkPos := TRUE;
		ELSE
			q_bWorkPos := FALSE;
		END_IF
	1:	(*If an error occurs, it gets controlled to the previous way, then releases the order*)
		IF (bEn AND bBaseposCmd AND (NOT bEHA OR NOT bError))
			OR (bEn AND bWorkPosCmd AND bEHA AND bErrWorkPos1 AND NOT i_bBasePos) THEN
			q_bBasePos := TRUE;
		ELSE
			q_bBasePos := FALSE;
		END_IF
		IF bEn AND bWorkPosCmd AND (NOT bEHA OR NOT bError)
			OR (bEn AND bBasePosCmd AND bEHA AND bErrBasePos1 AND NOT i_bWorkPos) THEN
			q_bWorkPos := TRUE;
		ELSE
			q_bWorkPos := FALSE;
		END_IF
	2:	(*No change control if an error occurs*)
		IF bEn AND bBaseposCmd THEN
			q_bBasePos := TRUE;
		ELSE
			q_bBasePos := FALSE;
		END_IF
		IF bEn  AND bWorkPosCmd THEN
			q_bWorkPos := TRUE;
		ELSE
			q_bWorkPos := FALSE;
		END_IF
END_CASE

(*Base position stabil*)
tBPS(IN:= q_bBasePos AND i_bBasePos AND NOT bError, PT:= timBasePosStab, Q=>  bBasePosStab);

(*Work position stabil*)
tWPS(IN:= q_bWorkPos AND i_bWorkPos AND NOT bError, PT:= timWorkPosStab, Q=>  bWorkPosStab);

(*Error string*)
IF bErrBasePos0 OR bErrBasePos1 OR bErrWorkPos0 OR bErrWorkPos1 OR bErrBPWP THEN
	sError := sName;
	IF bErrBasePos0 THEN
		sError := CONCAT(sError, CONCAT(' Base position error: the signal did not stop after reaching work position ', sBasePosSensor));
	END_IF
	IF bErrBasePos1 THEN
		sError := CONCAT(sError, CONCAT(' Base position error 1: the signal did not appear while reaching base position ', sBasePosSensor));
	END_IF
	IF bErrWorkPos0 THEN
		sError := CONCAT(sError,  CONCAT(' Work position error 0: the signal did not stop after reaching Work position ', sWorkPosSensor));
	END_IF
	IF bErrWorkPos1 THEN
		sError := CONCAT(sError, CONCAT(' Work position error 1: the signal did not appear while reaching work position ', sWorkPosSensor));
	END_IF
	IF bErrBPWP THEN
		sError := CONCAT(sError, CONCAT(' To positions at the same time error ', CONCAT(sBasePosSensor, CONCAT('-',sWorkPosSensor))));
	END_IF
ELSE
	sError := '';
END_IF

//Error clear
IF fbBasePosAlarm.eConfirmationState = 3 AND NOT bError THEN
	fbBasePosAlarm.Clear(0, FALSE);
END_IF	
IF fbWorkPosAlarm.eConfirmationState = 3 AND NOT bError THEN
	fbWorkPosAlarm.Clear(0, FALSE);
END_IF

END_FUNCTION_BLOCK

// ---- POUs/FBs/BTL/FB_BTL1AR0.TcPOU
FUNCTION_BLOCK FB_BTL1AR0
VAR_OUTPUT
	bValid					: BOOL;
	nDistance				: REAL;
END_VAR
VAR
	arrRaw		AT %I*		: ARRAY [0..3] OF BITARR8;
	nState		AT %I*		: USINT;
	nDword					: DINT;
	uConv2Dint				: U_to_dint;
	tValid					: TON;
	bDataValid				: BOOL;
END_VAR

uConv2Dint.arrRaw[0] := arrRaw[3];
uConv2Dint.arrRaw[1] := arrRaw[2];
uConv2Dint.arrRaw[2] := arrRaw[1];
uConv2Dint.arrRaw[3] := arrRaw[0];
IF uConv2Dint.nData <> 2147483647 AND nState = 3 THEN
	bDataValid := TRUE;
	nDistance := DINT_TO_REAL(uConv2Dint.nData)/1000;
ELSE
	bDataValid := FALSE;
	nDistance := 0;
END_IF

tValid(IN:= bDataValid, PT:= T#1S, Q=> bValid, ET=> );

END_FUNCTION_BLOCK

// ---- POUs/FBs/ServoVise/FB_ServoVise.TcPOU
FUNCTION_BLOCK FB_ServoVise
VAR_INPUT
	bErrorAck				: BOOL;
	bEnable					: BOOL;
	eCommand				: E_ServoVise_Command;
	bManualMode				: BOOL;
	lrTargetDistance		: LREAL;			// [mm]		Target distance without torque limit
	lrVisePosition			: LREAL;			// [mm]		Value of distance sensor
	bVisePosValid			: BOOL;				// []		Distane sensor status
	nTargetVelocity			: LREAL;			// [mm/s]
	nTorque					: LREAL := 20.0;	// [Nm]
	nTorqueRamp				: LREAL := 10.0;	// [%/s]
	nTorqueVelocityLimit	: LREAL := 0.1;		// [mm/s]
	nOverride				: LREAL := 100.0;	// [%] 
	nAttachVelocity			: LREAL := 0.1;
	nCalOffset_1			: LREAL := 22.32;
	nCalOffset_2			: LREAL := 99.01;
	nOpenOffset				: LREAL := 4;
	eViseJawState			: E_ViseJawState := E_ViseJawState.P1_0_120;
	stAxisEvent				: TcEventEntry;	(*Event definition*)
END_VAR
VAR_OUTPUT
	bReady					: BOOL;
	bBusy 					: BOOL;
	bDone 					: BOOL;
	bError 					: BOOL;
END_VAR
VAR (* Drive *)
	Axis					: AXIS_REF;
	fbPower					: MC_Power;
	fbMoveRelative			: MC_MoveRelative;
	fbReadDriveOpMode		: MC_ReadDriveOperationMode;
	fbWriteDriveOpMode		: MC_WriteDriveOperationMode;
	fbStop					: MC_Halt;
	fbHalt					: MC_Stop;
	fbTorqueControl			: MC_TorqueControl;	
	fbJog					: MC_Jog;
	fbTorqueCheck			: FB_TorqueCheck;	

	fbSoEReset				: FB_SoEReset;
	fbReset					: MC_Reset;
END_VAR
VAR (* State control *)
	nState 					: UDINT;
	nLastState				: UDINT;
	sState					: STRING;
	nTorqueRelief			: LREAL := 0.005;	// 0.005mm = 0.9°
	
	// Error control
	bIsInitalized			: BOOL;
	fbAlarm					: FB_TcAlarm;
	nGlobalAxisErrorID		: UDINT;
	
	//LastStates
	anLastStates			: ARRAY[0..500] OF UDINT;
    iLastStates				: INT;
	nRealVisePos			: LREAL;
END_VAR
VAR CONSTANT									//																			%     Tmax    i   Theta															
	nTScale					: LREAL := 2.3923;	// nTorque[Nm] / nTScale[Nm/%] = Required_torque_value[%]		{nTScale = 0.01 * 5.09 * 50 * 0.94}
END_VAR

(* Timers **************************************)

(* Enable **************************************)
IF NOT bEnable THEN
	fbPower.Enable := FALSE;
	fbTorqueControl.Execute := FALSE;
	fbMoveRelative.Execute := FALSE;
	nState := 0;
END_IF

(* States **************************************)
IF nLastState <> nState THEN
	nLastState := nState;
END_IF

(* State history ************************************************)
IF(nState >= 100) AND (nState <= 100000) THEN
(*Steps before any state*)
	IF anLastStates[0] <> nState THEN
		FOR iLastStates:=500 TO 1 BY -1 DO
			anLastStates[iLastStates]:= anLastStates[iLastStates-1];
		END_FOR
		anLastStates[0]:= nState;
	END_IF
END_IF	

(* Manual mode **************************************)
IF bManualMode THEN
	nState := 150000;
END_IF

(*Calculate Vise position **************************************)
IF eViseJawState = E_ViseJawState.P1_0_120 THEN
	nRealVisePos := lrVisePosition + nCalOffset_1;
ELSE
	nRealVisePos := lrVisePosition + nCalOffset_2;
END_IF

(* Error handling Tc3_EventLogger *******************************)
IF NOT bIsInitalized THEN
	bIsInitalized  :=  TRUE;
	fbAlarm.CreateEx(stAxisEvent, TRUE, 0);
END_IF

(* Error acknoledge **************************************)
IF bErrorAck THEN
	IF fbAlarm.eConfirmationState = 2 THEN
		fbAlarm.Confirm(0);
	END_IF
END_IF

IF Axis.Status.Error OR Axis.Status.DriveDeviceError OR fbPower.Error OR fbMoveRelative.Error OR fbTorqueControl.Error OR
	fbJog.Error OR fbSoEReset.Error OR fbReset.Error OR fbHalt.Error OR fbStop.Error OR fbReadDriveOpMode.Error OR fbWriteDriveOpMode.Error
THEN
	bError  :=  TRUE;
	IF (fbAlarm.eConfirmationState <> 2 AND fbAlarm.nTimeCleared <> 0 AND fbAlarm.nTimeConfirmed <> 0) OR //Ha már volt alarm, akkor van bennük érték
		(fbAlarm.eConfirmationState = 1 AND fbAlarm.nTimeCleared = 0 AND fbAlarm.nTimeConfirmed = 0)	//Első futás esetén
	THEN
		//fb_DriveDiag(Execute :=  TRUE, Axis :=  Axis);
		//IF NOT fb_DriveDiag.Busy THEN
			//fb_DriveDiag(Execute :=  FALSE, Axis :=  Axis);
			IF Axis.Status.ErrorID <> 0 THEN
				nGlobalAxisErrorID  :=  Axis.Status.ErrorID;
			ELSIF fbPower.ErrorID <> 0 THEN
				nGlobalAxisErrorID  :=  fbPower.ErrorID;
			ELSIF fbMoveRelative.ErrorID <> 0 THEN
				nGlobalAxisErrorID  :=  fbMoveRelative.ErrorID;
			ELSIF fbTorqueControl.ErrorID <> 0 THEN
				nGlobalAxisErrorID  :=  fbTorqueControl.ErrorID;
			ELSIF fbJog.ErrorID <> 0 THEN
				nGlobalAxisErrorID  :=  fbJog.ErrorID;
			ELSIF fbSoEReset.SercosErrId <> 0 THEN
				nGlobalAxisErrorID  :=  fbSoEReset.SercosErrId;
			ELSIF fbReset.ErrorID <> 0 THEN
				nGlobalAxisErrorID  :=  fbReset.ErrorID;
			END_IF
			//fbAlarm.ipArguments.Clear().AddUDInt(nGlobalAxisErrorID).AddUDInt(fb_DriveDiag.DiagNumber);
			fbAlarm.ipArguments.Clear().AddUDInt(nGlobalAxisErrorID);
			fbAlarm.Raise(0);
		//END_IF
	END_IF
END_IF

Axis();

CASE nState OF
{region "Alaphelyzet felvétel"}
	(****************************************************************************************)
	(******************************* Alaphelyzetfelvétel ************************************)
	(****************************************************************************************)	
	0:		(*-----=== Kimenetek törlése ===-----*)
		fbPower.Enable := FALSE;
		fbReadDriveOpMode.Execute := FALSE;
		fbWriteDriveOpMode.Execute := FALSE;
		fbStop.Execute := FALSE;
		fbHalt.Execute := FALSE;
		fbTorqueControl.Execute := FALSE;
		fbMoveRelative.Execute := FALSE;
		bBusy := FALSE;
		bDone := FALSE;
		bError := FALSE;
		IF bEnable THEN
			nState := nState + 20;
		END_IF
		
	20:		(*-----=== Axis és Drive hibák ellenőrzése ===-----*)
		IF Axis.Status.Error OR Axis.Status.DriveDeviceError THEN
			nState := 250000;
		ELSIF bEnable THEN
			nState := nState + 20;
		END_IF

	40:		(*-----=== Drive Op. mód ellenörzés ===-----*)
		fbReadDriveOpMode.Execute := TRUE;
		IF fbReadDriveOpMode.Done THEN
			IF fbReadDriveOpMode.DriveOperationMode <> Tc2_MC2.E_DriveOperationMode.DriveOperationMode_Default THEN
				nState := 10000;
			ELSE
				nState := 100;
			END_IF
			fbReadDriveOpMode.Execute := FALSE;
		END_IF

	100:		(*-----=== Drive átkapcsolása PtP módba ===-----*)
		fbWriteDriveOpMode.DriveOperationMode := Tc2_MC2.E_DriveOperationMode.DriveOperationMode_Default;
		fbWriteDriveOpMode.Execute := TRUE;
		IF fbWriteDriveOpMode.Done THEN
			fbWriteDriveOpMode.Execute := FALSE;
			nState := 10000;
		END_IF
{endregion}

{region "Alaphelyzet"}
	(****************************************************************************************)
	(*********************************** Alaphelyzet ****************************************)
	(****************************************************************************************)	
	10000:		(*-----=== Várakozás parancsra ===-----*)
		bReady := TRUE;
		bBusy := FALSE;
		bDone := FALSE;
		IF eCommand = E_ServoVise_Command.Fix THEN				// Nyomatékra húzás
			bBusy := TRUE;
			nState := 20000;
		ELSIF eCommand = E_ServoVise_Command.MoveToPos THEN		// Pozícionálás
			bBusy := TRUE;
			nState := 40000;
		ELSIF eCommand = E_ServoVise_Command.Release THEN		// Kioldás
			bBusy := TRUE;
			nState := 60000;
		ELSIF eCommand = E_ServoVise_Command.Attach THEN		// Tengelykapcsoló csatlakoztatása
			bBusy := TRUE;
			nState := 80000;
		END_IF
{endregion}

{region "Satu nyomatékrahúzása"}
	(****************************************************************************************)
	(****************************** Satu nyomatékrahúzás ************************************)
	(****************************************************************************************)	
	20000:		(*-----=== Szervo BE ===-----*)
		fbPower.Enable := TRUE;
		IF fbPower.Status THEN
			nState := 20100;
		ELSIF fbPower.Error THEN
			IF bStepEnable THEN
				nState := 250000;
			END_IF
		END_IF	
		
	20100:		(*-----=== Zárás nyomatékra ===-----*)
		fbTorqueControl.Torque := -1 * ABS(nTorque/nTScale);					// Nyomaték átszámítása Nm-ből %-ba
		fbTorqueControl.TorqueRamp := nTorqueRamp;
		fbTorqueControl.VelocityLimitHigh := nTorqueVelocityLimit;
		fbTorqueControl.VelocityLimitLow := -1 * nTorqueVelocityLimit;
		fbTorqueControl.Execute := TRUE;
		IF fbTorqueControl.Busy THEN
			IF bStepEnable THEN
				nTorqueRelief := ((ABS(nTorque))/6000 + (1/300));					// A feszültségmentesítési szög nyomatékfüggő!! Y=m*X+b	{m=1/6000, b=1/300}
				nState := nState + 20;
			END_IF
		END_IF
	
	20120:		(*-----=== Nyomaték figyelés ===-----*)
		IF fbTorqueCheck.bTorqueDone THEN
			IF bStepEnable THEN
				fbTorqueControl.Execute := FALSE;
				nState := nState + 20;
			END_IF
		ELSIF fbTorqueControl.Error THEN
			nState := 250000;
		ELSIF (lrVisePosition < 0) AND bVisePosValid THEN						// Minimális pozíció elérve -> Hiba
			nState := 250000;
		ELSIF (nRealVisePos < (lrTargetDistance - 6)) THEN						// Satupozíció 4mm-el kissebb mint a nominál méret -> Hiba
			nState := 250000;
		END_IF	
	
	20140:		(*-----=== Axis Halt ===-----*)(*-----=== Váratla mozgások elkerülése ===-----*)
		fbHalt.Execute := TRUE;
		IF fbHalt.Done THEN
			IF bStepEnable THEN
				fbHalt.Execute := FALSE;
				nState:= nState + 20;
			END_IF
		END_IF
	
	20160:		(*-----=== Átkapcsolás pozíció módba ===-----*)
		fbWriteDriveOpMode.DriveOperationMode := Tc2_MC2.E_DriveOperationMode.DriveOperationMode_Default;
		fbWriteDriveOpMode.Execute := TRUE;
		IF fbWriteDriveOpMode.Done THEN
			IF bStepEnable THEN
				fbWriteDriveOpMode.Execute := FALSE;
				nState := nState + 20;
			END_IF
		END_IF
	
	20180:		(*-----=== Szervo Mozgatás PtP ===-----*)
		fbMoveRelative.Distance := 0.055;(*nTorqueRelief*) //New clutch based on appx. 10 degree, counted with 2mm slope of shaft
		fbMoveRelative.Velocity := nTargetVelocity;
		fbMoveRelative.Execute := TRUE;
		IF fbMoveRelative.Done THEN
			IF bStepEnable THEN
				fbMoveRelative.Execute := FALSE;
				nState := nState + 20;
			END_IF
		ELSIF fbMoveRelative.Error THEN
			fbMoveRelative.Execute := FALSE;
			nState := 250000;
		END_IF
	
	20200:		(*-----=== Szervo KI ===-----*)
		fbPower.Enable := FALSE;
		nState := nState + 20;
	
	20220:		(*-----=== Várakozás parancs törlésre ===-----*)
		bBusy := FALSE;
		bDone := TRUE;
		IF eCommand = E_ServoVise_Command.NoCommand THEN
			IF bStepEnable THEN
				nState := 10000;
			END_IF
		END_IF
{endregion}

{region "Satu pzícionálás"}
	(****************************************************************************************)
	(********************************* Satu pozícionálás ************************************)
	(****************************************************************************************)	
	40000:		(*-----=== Szervo BE ===-----*)
		fbPower.Enable := TRUE;
		IF fbPower.Status THEN
			nState := nState + 20;
		ELSIF fbPower.Error THEN
			nState := 250000;
		END_IF
			
	40020:		(*-----=== Szervo Mozgatás PtP ===-----*)
		fbMoveRelative.Distance := (lrTargetDistance + nOpenOffset) - nRealVisePos;
		fbMoveRelative.Velocity := nTargetVelocity;
		fbMoveRelative.Execute := TRUE;
		IF fbMoveRelative.Done THEN
			IF bStepEnable THEN
				fbMoveRelative.Execute := FALSE;
				nState := nState + 20;
			END_IF
		ELSIF fbMoveRelative.Error THEN
			fbMoveRelative.Execute := FALSE;
			nState := 250000;
		ELSIF (lrVisePosition < 0) AND bVisePosValid AND fbMoveRelative.Distance < 0 THEN						// Minimális pozíció elérve -> Hiba
			nState := 250000;
		ELSIF (lrVisePosition > 125) AND bVisePosValid AND fbMoveRelative.Distance > 0 THEN						// Maximális pozíció elérve -> Hiba
			nState := 250000;
		END_IF
		
	40040:		(*-----=== Szervo KI ===-----*)
		fbPower.Enable := FALSE;
		nState := nState + 20;
	
	40060:		(*-----=== Várakozás parancs törlésre ===-----*)
		bBusy := FALSE;
		bDone := TRUE;
		IF eCommand = E_ServoVise_Command.NoCommand THEN
			IF bStepEnable THEN
				nState := 10000;
			END_IF
		END_IF
{endregion}

{region "Satu oldása"}
	(****************************************************************************************)
	(************************************ Satu elengedés ************************************)
	(****************************************************************************************)
	60000:		(*-----=== Szervo BE ===-----*)
		fbPower.Enable := TRUE;
		IF fbPower.Status THEN
			nState := nState + 20;
		ELSIF fbPower.Error THEN
			nState := 250000;
		END_IF
	
	60020:		(*-----=== Szervo Mozgatás PtP ===-----*)
		fbMoveRelative.Distance := nOpenOffset;
		fbMoveRelative.Velocity := nTargetVelocity;
		fbMoveRelative.Execute := TRUE;
		IF fbMoveRelative.Done THEN
			IF bStepEnable THEN
				fbMoveRelative.Execute := FALSE;
				nState := nState + 20;
			END_IF
		ELSIF fbMoveRelative.Error THEN
			fbMoveRelative.Execute := FALSE;
			nState := 250000;
		END_IF
	
	60040:		(*-----=== Szervo KI ===-----*)
		fbPower.Enable := FALSE;
		nState := nState + 20;
		
	60060:		(*-----=== Várakozás parancs törlésre ===-----*)
		bBusy := FALSE;
		bDone := TRUE;
		IF eCommand = E_ServoVise_Command.NoCommand THEN
			IF bStepEnable THEN
				nState := 10000;
			END_IF
		END_IF
{endregion}

{region "Satu csatlakoztatása"}
	(****************************************************************************************)
	(********************************** Satu csatlakoztatás *********************************)
	(****************************************************************************************)
	80000:		(*-----=== Szervo BE ===-----*)
		fbPower.Enable := TRUE;
		IF fbPower.Status THEN
			nState := nState + 20;
		ELSIF fbPower.Error THEN
			nState := 250000;
		END_IF	
		
	80020:		(*-----=== Zárás nyomatékra ===-----*)
		fbTorqueControl.Torque := -5;
		fbTorqueControl.TorqueRamp := nTorqueRamp;
		fbTorqueControl.VelocityLimitHigh := nAttachVelocity;
		fbTorqueControl.VelocityLimitLow := -1 * nAttachVelocity;
		fbTorqueControl.Execute := TRUE;
		IF fbTorqueControl.Busy THEN
			IF bStepEnable THEN
				nState := nState + 20;
			END_IF
		END_IF
	
	80040:		(*-----=== Várakozás parancs törlésre ===-----*)
		bBusy := FALSE;
		bDone := TRUE;
		IF eCommand = E_ServoVise_Command.NoCommand THEN
			IF bStepEnable THEN
				fbTorqueControl.Execute := FALSE;
				nState:= nState + 20;
			END_IF
		END_IF
	
	80060:		(*-----=== Axis Halt ===-----*)(*-----=== Váratla mozgások elkerülése ===-----*)
		fbHalt.Execute := TRUE;
		IF fbHalt.Done THEN
			IF bStepEnable THEN
				fbHalt.Execute := FALSE;
				nState:= nState + 20;
			END_IF
		END_IF
	
	80080:		(*-----=== Átkapcsolás pozíció módba ===-----*)
		fbWriteDriveOpMode.DriveOperationMode := Tc2_MC2.E_DriveOperationMode.DriveOperationMode_Default;
		fbWriteDriveOpMode.Execute := TRUE;
		IF fbWriteDriveOpMode.Done THEN
			IF bStepEnable THEN
				fbWriteDriveOpMode.Execute := FALSE;
				nState := nState + 20;
			END_IF
		END_IF
	
	80100:		(*-----=== Szervo KI ===-----*)
		fbPower.Enable := FALSE;
		nState := 10000;
{endregion}

{region "Manual mód"}
	(****************************************************************************************)
	(*************************************** Kézi üzem **************************************)
	(****************************************************************************************)	
	150000:		(*-----=== Manual mode ===-----*)
		fbJog.Mode := MC_JOGMODE_CONTINOUS;
		IF NOT bManualMode THEN
			nState := 10000;
		END_IF
		IF fbJog.Error THEN
			nState := 250000;
		END_IF
{endregion}

{region "Hibakezelés"}
	(****************************************************************************************)
	(************************************* Hibakezelés **************************************)
	(****************************************************************************************)	
	250000:		(*-----=== Error ===-----*)
		bReady := FALSE;
		bBusy := FALSE;
		bDone := FALSE;
		bError := TRUE;
		fbReadDriveOpMode.Execute := FALSE;
		fbWriteDriveOpMode.Execute := FALSE;
		fbStop.Execute := FALSE;
		fbHalt.Execute := FALSE;
		fbTorqueControl.Execute := FALSE;
		fbMoveRelative.Execute := FALSE;
		IF Axis.Status.HasJob THEN
			nState := nState + 20;
		ELSE
			nState := nState + 40;
		END_IF
	
	250020:	(* Axis halt *)
		fbHalt.Execute := TRUE;
		IF fbHalt.Done THEN
			IF bStepEnable THEN
				fbHalt.Execute := FALSE;
				nState:= nState + 20;
			END_IF
		END_IF
	
	250040: (*Wait error ACK*)
		IF bErrorAck THEN
			nState := nState + 20;
		END_IF
		
	250060: (*Error ACK*)
		IF Axis.Status.DriveDeviceError THEN
			IF bStepEnable THEN 
				fbSoEReset.Execute := TRUE;
				fbReset.Execute := TRUE;
				nState := 250080;
			END_IF
		ELSIF Axis.Status.Error THEN
			IF bStepEnable THEN 
				fbReset.Execute := TRUE;
				nState := 250100;
			END_IF
		ELSE
			nState := 0;
		END_IF
		
	250080: (*Drive Reset*)
		IF NOT fbSoEReset.Busy THEN
			fbSoEReset.Execute := FALSE;
			nState := 0;
		ELSIF fbSoEReset.Error THEN
			nState := 0; 
		END_IF
		
	250100: (*Reset*)
		IF fbReset.Done THEN
			fbReset.Execute := FALSE;
			nState := 0;
		ELSIF fbReset.Error THEN
			nState := 0; 
		END_IF	
{endregion}
ELSE
	sState := 'Not used step';	
END_CASE


ActPower();
ActHalt();
ActStop();
ActMode();
ActTorque();
ActMoveRelative();
ActJog();
ActSoEReset();
ActReset();

ACTION ActHalt:
fbHalt(Axis:= Axis);
END_ACTION

ACTION ActJog:
fbJog(
	Axis:= Axis, 
	JogForward:= TRUE, 
	JogBackwards:= TRUE, 
	Mode:= fbJog.Mode, 
	Velocity:= 10);
END_ACTION

ACTION ActMode:
fbReadDriveOpMode(
	Axis:= Axis, 
	Execute:= , 
	Options:= , 
	Done=> , 
	Busy=> , 
	Error=> , 
	ErrorID=> , 
	DriveOperationMode=> );

fbWriteDriveOpMode(
	Axis:= Axis, 
	Execute:= , 
	DriveOperationMode:= , 
	Options:= , 
	Done=> , 
	Busy=> , 
	Error=> , 
	ErrorID=> );
END_ACTION

ACTION ActMoveRelative:
fbMoveRelative(
	Axis:= Axis);
//, 
//	Distance:= lrCalculatedDistance, 
//	Velocity:= nOpenVelocity);
END_ACTION

ACTION ActPower:
fbPower(
	Axis:= Axis, 
	Enable_Positive:= TRUE, 
	Enable_Negative:= TRUE, 
	Override:= nOverride);
END_ACTION

ACTION ActReset:
fbReset(Axis:= Axis);
END_ACTION

ACTION ActSoEReset:
fbSoEReset(Axis:= Axis);
END_ACTION

ACTION ActStop:
fbStop(Axis:= Axis);
END_ACTION

ACTION ActTorque:
fbTorqueControl(
	Axis:= Axis, 
	ContinuousUpdate:= FALSE, 
	Relative:= FALSE, 
	Torque:= , 
	TorqueRamp:= , 
	VelocityLimitHigh:= , 
	VelocityLimitLow:= );

fbTorqueCheck(
	Axis:= Axis, 
	bEnable:= fbTorqueControl.Execute, 
	nTorque:= fbTorqueControl.Torque, 
	tTorqueStabTime:= T#500ms, 
	bTorqueDone=> );
END_ACTION

END_FUNCTION_BLOCK

// ---- POUs/FBs/ServoVise/FB_TorqueCheck.TcPOU
FUNCTION_BLOCK FB_TorqueCheck
VAR_IN_OUT
    Axis 					: AXIS_REF;
END_VAR
VAR_INPUT
	bEnable					: BOOL;
	nTorque					: LREAL;
	tTorqueStabTime			: TIME := T#500ms;
END_VAR
VAR_OUTPUT
	bTorqueDone				: BOOL;
END_VAR
VAR
	bAxisNotMove			: BOOL;
	timNotMove				: TON;
	bAxisInTorque			: BOOL;
	timInTorque				: TON;
	timStab					: TON;
END_VAR

timNotMove(IN:= ABS(Axis.NcToPlc.ActVelo)<0.01, PT:= T#200ms, Q=> bAxisNotMove, ET=> );
timInTorque(IN:= ABS(ABS(Axis.NcToPlc.ActTorque) - ABS(nTorque))< 3, PT:= T#200ms, Q=>bAxisInTorque , ET=> );
timStab(IN:= bAxisNotMove AND bAxisInTorque, PT:= tTorqueStabTime, Q=> , ET=> );
bTorqueDone := timStab.Q AND bEnable;

END_FUNCTION_BLOCK

// ---- POUs/CNC_2/CNC_2.TcPOU
PROGRAM CNC_2
VAR	(* Control *)
	nState						: UDINT;
	nStatePrevious				: UDINT;
	sState						: STRING(500);
	fbCycleTime					: TON;
	nCycleTime					: REAL;
	bError						: BOOL;
END_VAR
VAR (* LastStates *)
	anLastStates				: ARRAY[0..500] OF UDINT;
    iLastStates					: INT;
END_VAR
VAR (* Var IO *)
	{attribute 'TcLinkTo' := '		.fbMoveUpper.i_bBasePos	:= TIIB(24)^Channel 1^Input;
									.fbMoveUpper.i_bWorkPos	:= TIIB(24)^Channel 2^Input;
									.fbMoveUpper.q_bBasePos	:= TIIB(25)^Channel 2^Output;
									.fbMoveUpper.q_bWorkPos	:= TIIB(25)^Channel 1^Output;
									.fbMoveLower.i_bBasePos	:= TIIB(24)^Channel 3^Input;
									.fbMoveLower.i_bWorkPos	:= TIIB(24)^Channel 4^Input;
									.fbMoveLower.q_bBasePos	:= TIIB(25)^Channel 4^Output;
									.fbMoveLower.q_bWorkPos	:= TIIB(25)^Channel 3^Output;
									.fbLock.i_bBasePos	:= TIIB(24)^Channel 6^Input;
									.fbLock.i_bWorkPos	:= TIIB(24)^Channel 5^Input;
									.fbLock.q_bWorkPos	:= TIIB(25)^Channel 5^Output;
									.q_bToolCheckBlower := TIIB(25)^Channel 6^Output;
									.fbVisePos.arrRaw[0]	:= TIIB(21)^Module 1 (IOL_I_4byte)^TxPDO^input byte 0;	
									.fbVisePos.arrRaw[1] 	:= TIIB(21)^Module 1 (IOL_I_4byte)^TxPDO^input byte 1;
									.fbVisePos.arrRaw[2]	:= TIIB(21)^Module 1 (IOL_I_4byte)^TxPDO^input byte 2;
									.fbVisePos.arrRaw[3]	:= TIIB(21)^Module 1 (IOL_I_4byte)^TxPDO^input byte 3;
									.fbVisePos.nState		:= TIIB(21)^IO-Link DeviceState Inputs^Status of IO-Link Port 1;'}
	fbCncServoVise				: FB_CNC_Servo;	

END_VAR
VAR (* OPC_UA *)
	stCNC_Data					: 	POINTER TO OPC_CNC_Data_Collection;
	tHeartBeatDelay				: 	TON;
	bCNCHandshakeTimeout		:	BOOL;
	tCNCHandshakeTimer			:	TON;
	bCNCMidwareShutdownPossible	: 	BOOL;	//20, 40, 11400, 
	bShutdownIsProcessing		:	BOOL;
END_VAR
VAR (*Test components*)
	bEnableStart				:	BOOL := FALSE;
END_VAR
VAR	(*7 Axis Robot Communication*)
	bCNCRunning					:	BOOL;
END_VAR

(* OPC_UA *)
stCNC_Data := ADR(OPC_UA_CNC2);
tHeartBeatDelay(IN := stCNC_Data^.HeartBeat = 99, PT := T#500MS, Q=>);
IF tHeartBeatDelay.Q THEN
	stCNC_Data^.HeartBeat := 0;
END_IF

tCNCHandshakeTimer(		IN :=	(stCNC_Data^.HeartBeat = 0),
						PT := T#3S,
						Q=>bCNCHandshakeTimeout);
					
					
(* =================================== OPC_UA Automatic Shutdown handling =========================================== *)					
bCNCMidwareShutdownPossible := 	nState <= 10000;
								
IF bCNCMidwareShutdownPossible AND stCNC_Data^.MidwareRequestedShutdown AND (NOT bCNCHandshakeTimeout) THEN
	stCNC_Data^.ApproveShutdownRequest := TRUE;
END_IF

IF stCNC_Data^.ApproveShutdownRequest THEN
	IF bCNCHandshakeTimeout THEN
		bShutdownIsProcessing := TRUE;
	END_IF
END_IF

IF bShutdownIsProcessing THEN
	stCNC_Data^.ApproveShutdownRequest := FALSE;
	stCNC_Data^.MidwareRequestedShutdown := FALSE;
	IF (NOT bCNCHandshakeTimeout) THEN
		bShutdownIsProcessing := FALSE;
	END_IF
END_IF

(*Error handling*)
IF nState > 0 AND nState < 150000 THEN
	nStatePrevious := nState;
END_IF

(*Maintance*)
IF bManualMode THEN
	nState := 150000;
END_IF

(*Emergency*)
IF NOT i_bLO1_Main THEN
	nState := 0;
END_IF

(*Last states*)
IF(nState >= 1000) AND (nState < 150000) THEN
(*Steps before any state*)
	IF anLastStates[0] <> nState THEN
		FOR iLastStates:=500 TO 1 BY -1 DO
			anLastStates[iLastStates]:= anLastStates[iLastStates-1];
		END_FOR
		anLastStates[0]:= nState;
	END_IF
END_IF	

IF fbCncServoVise.bError (*OR stCNC_Data^.ControlStatus_Error*)
THEN
	bError  :=  TRUE;
END_IF


(*   Vise Position Adjustment  -16,38 *)
fbCncServoVise.nCalOffset_1 := 14.94;	//Originally 22.32
fbCncServoVise.nCalOffset_2 := 91.63;	//Originally 99.01

bCNCRunning := ((nState > 10000) AND (nState <= 30000));

CASE nState OF
{region "Alaphelyzet felvétel"}
	(****************************************************************************************)
	(******************************* Alaphelyzetfelvétel ************************************)
	(****************************************************************************************)	
	0:		(*-----=== Kimenetek törlése ===-----*)
		sState := CONCAT(UDINT_TO_STRING(nState) ,' - A biztonsági kör nem aktív');
		IF i_bLO1_Main AND (NOT bManualMode) THEN		//AND i_bLO1_CNC1 THEN		Nincs bekötve! Teszteléshez kikapcsolva! Ha a bekötés kész VISSZAÍRNI !!!!!!!!!!!!!!!
			stCNC_Data^.DoorControl_CloseDoor := FALSE;
			stCNC_Data^.DoorControl_OpenDoor := FALSE;
			stCNC_Data^.MagazineTable_Trigger := FALSE;
			stCNC_Data^.ToolTable_Trigger := FALSE;
			stCNC_Data^.M401_Acknowledge := FALSE;
			stCNC_Data^.M402_Acknowledge := FALSE;
			stCNC_Data^.M403_Acknowledge := FALSE;
			stCNC_Data^.StartCNCProgram := FALSE;
			stCNC_Data^.StopCNCProgram := FALSE;
			stCNC_Data^.CancelCNCProgram := FALSE;
			stCNC_Data^.SelectCNCProgramByNodeID := FALSE;
			stCNC_Data^.SelectCNCPrograBlockNumber := FALSE;
//			stCNC_Data^.ToolTablePath := '';
			stCNC_Data^.ToolTableLoadTrigger := FALSE;
			stCNC_Data^.MagazineTableLoadTrigger := FALSE;
			stCNC_Data^.ProgramLoadTrigger := FALSE;
			IF bStepEnable THEN
				nState := nState + 20;
			END_IF
		END_IF

	20:		(*-----=== CNC ellenőrzés ===-----*)
		sState := CONCAT(UDINT_TO_STRING(nState) ,' - A CNC ellenőrzése');
		IF stCNC_Data^.ServerState = 'Running' AND
		   stCNC_Data^.CurrentState_State = 'NCIsAvailable' THEN
				IF		stCNC_Data^.CurentState_Program = 'Running' THEN
					nState := 11500;										// A megmunkálás folyamatban -> Várakozás megmunkálás végére.
				ELSIF	stCNC_Data^.CurentState_Program = 'Idle' OR stCNC_Data^.CurentState_Program = 'NotSelected' OR stCNC_Data^.CurentState_Program = 'Interrupted' THEN
					IF (stDutData_Cnc2.nDutId > 0 AND stDutData_Cnc2.bDone) OR stDutData_Cnc2.bDutInVise THEN
						IF bStepEnable THEN									// Késztermék a satuban
							nState := 11560;
						END_IF
					ELSE
						IF bStepEnable THEN									// A satu üres
							nState := nState + 20;
						END_IF
					END_IF
				END_IF
		END_IF

	40:		(*-----=== CNC ajtó nnyitása ===-----*)
		sState := CONCAT(UDINT_TO_STRING(nState) ,' - A CNC ajtó nyitása');
		stCNC_Data^.DoorControl_OpenDoor := TRUE;
		IF stCNC_Data^.DoorControl_DoorOpened THEN
			IF bStepEnable THEN	
				stCNC_Data^.DoorControl_OpenDoor := FALSE;
				nState := nState + 20;
			END_IF
		END_IF

	60:
		nState := 10000;
{endregion}

{region "Alaphelyzet"}
	(****************************************************************************************)
	(*********************************** Alaphelyzet ****************************************)
	(****************************************************************************************)	
	10000:		(*-----=== Várakozás berakásra ===-----*)
		sState := CONCAT(UDINT_TO_STRING(nState) ,' - Várakozás alapanyagra');
		IF ((NOT bShutdownIsProcessing) AND (NOT stCNC_Data^.ApproveShutdownRequest)) THEN
			IF Robot7AxisProgram.bStartCNC2 THEN
				IF stDutData_Cnc2.nDutId > 0 THEN											// Alapanyag a robotnál
					IF bStepEnable THEN	
						nState := 11000;			// -> Alapanyag fogadása
					END_IF
				END_IF
			END_IF
		END_IF
{endregion}

{region "Alapanyag fogadása"}
	(****************************************************************************************)
	(******************************** Alapanyag fogadása ************************************)
	(****************************************************************************************)	
	11000:		(*-----=== Satu pozícionálása ===-----*)
		sState := CONCAT(UDINT_TO_STRING(nState) ,' - Satu pozícionálása');
		fbCncServoVise.nPosition := stDutData_Cnc2.nDimX;
		fbCncServoVise.eCommand := E_CncServoCommand.MovePos;
		IF fbCncServoVise.bDone THEN
			IF bStepEnable THEN
				fbCncServoVise.eCommand := E_CncServoCommand.NoCommand;
				nState := 11100;
			END_IF
		END_IF

	11100:		(*-----=== Várakozás alapanyag berakásra ===-----*)
		sState := CONCAT(UDINT_TO_STRING(nState) ,' - Alapanyag berakás');
		IF Robot7AxisProgram.fbRobot.bZoneCnc2 THEN
			IF bStepEnable THEN
				stDutData_Cnc2.bDutInVise := TRUE;
				nState := 11200;
			END_IF
		END_IF

	11200:		(*-----=== Várakozás robot távozásra ===-----*)
		sState := CONCAT(UDINT_TO_STRING(nState) ,' - Várakozás robot távozásra');
		IF NOT Robot7AxisProgram.fbRobot.bZoneCnc2 THEN
			IF bStepEnable THEN
				nState := 11300;
			END_IF
		END_IF
	
	11300:		(*-----=== Satu rögzítése ===-----*)
		sState := CONCAT(UDINT_TO_STRING(nState) ,' - Satu rögzítése');
		fbCncServoVise.nTorque := stDutData_Cnc2.nTorque;
		fbCncServoVise.eCommand := E_CncServoCommand.Fixed;
		IF fbCncServoVise.bDone THEN
			IF bStepEnable THEN
				fbCncServoVise.eCommand := E_CncServoCommand.NoCommand;
				nState := 11400;
			END_IF
		END_IF

	11400:		(*-----=== CNC ajtó zárása ===-----*)
		sState := CONCAT(UDINT_TO_STRING(nState) ,' - A CNC ajtó zárása');
		stCNC_Data^.DoorControl_CloseDoor := TRUE;
		IF stCNC_Data^.DoorControl_DoorClosed THEN
			IF bStepEnable THEN	
				stCNC_Data^.DoorControl_CloseDoor := FALSE;
				nState := nState + 20;
			END_IF
		END_IF

	11420:		(*-----=== CNC előkészítése ===-----*)
		sState := CONCAT(UDINT_TO_STRING(nState) ,' - A CNC előkészítése');
		IF TRUE THEN															// Külön FB-be rakni mert még képlékeny CAM file letöltése, ellenőrzése, felmásolása, betöltése, ........ 
			IF bStepEnable THEN	
				nState := nState + 20;
			END_IF
		END_IF

	11440:		(*-----=== CAM program indítása ===-----*)
		sState := CONCAT(UDINT_TO_STRING(nState) ,' - CAM program indítása');
		stCNC_Data^.StartCNCProgram := TRUE;
		IF stCNC_Data^.CurentState_Program = 'Running' THEN
			IF bStepEnable THEN	
				stCNC_Data^.StartCNCProgram := FALSE;
				nState := 11500;
			END_IF
		END_IF
	
	11500:		(*-----=== Várakozás CAM program végére ===-----*)
		sState := CONCAT(UDINT_TO_STRING(nState) ,' - Várakozás CAM program végére');
		IF stCNC_Data^.CurentState_Program = 'Finished' OR stCNC_Data^.CurentState_Program = 'Idle' THEN
			IF bStepEnable THEN	
				stCNC_Data^.DoorControl_CloseDoor := FALSE;
				nState := nState + 20;
			END_IF
		END_IF

	11520:		(*-----=== CNC folyamat befejezése ===-----*)
		sState := CONCAT(UDINT_TO_STRING(nState) ,' - A CNC folyamat befejezése');
		IF TRUE THEN															// Külön FB-be rakni mert még képlékeny: minőségellenőrzés, mérési adatok, .... 
			IF bStepEnable THEN	
				nState := nState + 20;
			END_IF
		END_IF

	11540:		(*-----=== CAM program leállítása ===-----*)
		sState := CONCAT(UDINT_TO_STRING(nState) ,' - CAM program leállítása');
		stCNC_Data^.CancelCNCProgram := TRUE;
		IF stCNC_Data^.CurentState_Program = 'Idle' THEN
			IF bStepEnable THEN	
				stCNC_Data^.CancelCNCProgram := FALSE;
				nState := nState + 20;
			END_IF
		END_IF

	11560:		(*-----=== CNC ajtó nnyitása ===-----*)
		sState := CONCAT(UDINT_TO_STRING(nState) ,' - A CNC ajtó nyitása');
		stCNC_Data^.DoorControl_OpenDoor := TRUE;
		IF stCNC_Data^.DoorControl_DoorOpened THEN
			IF bStepEnable THEN	
				stCNC_Data^.DoorControl_OpenDoor := FALSE;
				nState := 11600;
			END_IF
		END_IF
	
	11600:		(*-----=== Satu pozícionálása ===-----*)
		sState := CONCAT(UDINT_TO_STRING(nState) ,' - Satu pozícionálása');
		fbCncServoVise.nPosition := stDutData_Cnc2.nDimX;
		fbCncServoVise.eCommand := E_CncServoCommand.MovePos;
		IF fbCncServoVise.bDone THEN
			IF bStepEnable THEN
				stDutData_Cnc2.bDone := TRUE;
				stDutData_Cnc2.bPass := TRUE;
				fbCncServoVise.eCommand := E_CncServoCommand.NoCommand;
				nState := 12000;
			END_IF
		END_IF
{endregion}

{region "Alapanyag küldése"}
	(****************************************************************************************)
	(******************************** Alapanyag küldése ************************************)
	(****************************************************************************************)	
	12000:		(*-----=== Várakozás alapanyag kivételre ===-----*)
		sState := CONCAT(UDINT_TO_STRING(nState) ,' - Alapanyag kivétel');
		IF Robot7AxisProgram.fbRobot.bZoneCnc2 THEN
			IF bStepEnable THEN
				nState := 12100;
			END_IF
		END_IF
	
	12100:		(*-----=== Várakozás robot távozásra ===-----*)
		sState := CONCAT(UDINT_TO_STRING(nState) ,' - Satu rögzítése');
		IF NOT Robot7AxisProgram.fbRobot.bZoneCnc2 THEN
			IF bStepEnable THEN
				stDutData_Cnc2.bDutInVise := FALSE;
				stDutData_Cnc2.nDutId := 0;
				stDutData_Cnc2.bDone := FALSE;
				nState := 10000;
			END_IF
		END_IF
{endregion}

	150000: (* Maintenance *)
		sState := CONCAT(UDINT_TO_STRING(nState) ,' - Maintenance');
		IF NOT bManualMode THEN
			nState := 0;
		END_IF
		
	200000:(* Error handling *)
		sState := CONCAT(UDINT_TO_STRING(nState) ,CONCAT(' - Error, from this state: ' , sState));
		nState := 200020;

	200020:(* Error handling *)
		IF bAckP THEN
			CASE nStatePrevious OF
				0..9999: nState := 0;
//				10000..25000: nState := 10000;
//				30000..31000: nState := 30000;
			ELSE nState := 0;
			END_CASE
		END_IF	
		
	ELSE //Not a real step, for test purposes
		sState := CONCAT(UDINT_TO_STRING(nState) ,' - Not a real step, for test purposes');
END_CASE

(*Timers***************************************************)
fbCycleTime(IN:= nState > 10000 AND nState <= 95000, PT:= T#1D, Q=> , ET=> );
IF nState > 10000 AND nState <= 95000 THEN
	nCycleTime := TIME_TO_REAL(fbCycleTime.ET)/1000;
END_IF

ServoVise();
//fbCncServoVise.bTestUp := i_bTest_Up;
//fbCncServoVise.bTestDown := i_bTest_Down;
//fbCncServoVise.bTestStop := i_bTest_Stop;

ACTION ServoVise:
fbCncServoVise(
	sName:= 'AWEA_2', 
	bErrorAck:= bAckP, 
	bEnable:= i_bLO1_Main,		//AND i_bLO1_CNC1 THEN		Nincs bekötve! Teszteléshez kikapcsolva! Ha a bekötés kész VISSZAÍRNI !!!!!!!!!!!!!!!, 
	bManualMode:= bManualMode, 
	bReady=> , 
	bBusy=> , 
	bDone=> , 
	bError=> );
END_ACTION

END_PROGRAM

// ---- POUs/CNC_3/CNC_3.TcPOU
PROGRAM CNC_3
VAR	(* Control *)
	nState						: UDINT;
	nStatePrevious				: UDINT;
	sState						: STRING(500);
	fbCycleTime					: TON;
	nCycleTime					: REAL;
	bError						: BOOL;
END_VAR
VAR (* LastStates *)
	anLastStates				: ARRAY[0..500] OF UDINT;
    iLastStates					: INT;
END_VAR
VAR (* Var IO *)
	{attribute 'TcLinkTo' := '		.fbMoveUpper.i_bBasePos	:= TIIB(35)^Channel 1^Input;
									.fbMoveUpper.i_bWorkPos	:= TIIB(35)^Channel 2^Input;
									.fbMoveUpper.q_bBasePos	:= TIIB(36)^Channel 2^Output;
									.fbMoveUpper.q_bWorkPos	:= TIIB(36)^Channel 1^Output;
									.fbMoveLower.i_bBasePos	:= TIIB(35)^Channel 3^Input;
									.fbMoveLower.i_bWorkPos	:= TIIB(35)^Channel 4^Input;
									.fbMoveLower.q_bBasePos	:= TIIB(36)^Channel 4^Output;
									.fbMoveLower.q_bWorkPos	:= TIIB(36)^Channel 3^Output;
									.fbLock.i_bBasePos	:= TIIB(35)^Channel 6^Input;
									.fbLock.i_bWorkPos	:= TIIB(35)^Channel 5^Input;
									.fbLock.q_bWorkPos	:= TIIB(36)^Channel 5^Output;
									.q_bToolCheckBlower := TIIB(36)^Channel 6^Output;
									.fbVisePos.arrRaw[0]	:= TIIB(32)^Module 1 (IOL_I_4byte)^TxPDO^input byte 0;	
									.fbVisePos.arrRaw[1] 	:= TIIB(32)^Module 1 (IOL_I_4byte)^TxPDO^input byte 1;
									.fbVisePos.arrRaw[2]	:= TIIB(32)^Module 1 (IOL_I_4byte)^TxPDO^input byte 2;
									.fbVisePos.arrRaw[3]	:= TIIB(32)^Module 1 (IOL_I_4byte)^TxPDO^input byte 3;
									.fbVisePos.nState		:= TIIB(32)^IO-Link DeviceState Inputs^Status of IO-Link Port 1;'}
	fbCncServoVise				: FB_CNC_Servo;	

END_VAR
VAR (* OPC_UA *)
	stCNC_Data					: 	POINTER TO OPC_CNC_Data_Collection;
	tHeartBeatDelay				: 	TON;
	bCNCHandshakeTimeout		:	BOOL;
	tCNCHandshakeTimer			:	TON;
	bCNCMidwareShutdownPossible	: 	BOOL;	//20, 40, 11400, 
	bShutdownIsProcessing		:	BOOL;
END_VAR
VAR (*Test components*)
	bEnableStart				:	BOOL := FALSE;
END_VAR
VAR	(*7 Axis Robot Communication*)
	bCNCRunning					:	BOOL;
END_VAR

(* OPC_UA *)
stCNC_Data := ADR(OPC_UA_CNC3);
tHeartBeatDelay(IN := stCNC_Data^.HeartBeat = 99, PT := T#500MS, Q=>);
IF tHeartBeatDelay.Q THEN
	stCNC_Data^.HeartBeat := 0;
END_IF

tCNCHandshakeTimer(		IN :=	(stCNC_Data^.HeartBeat = 0),
						PT := T#3S,
						Q=>bCNCHandshakeTimeout);
					
					
(* =================================== OPC_UA Automatic Shutdown handling =========================================== *)					
bCNCMidwareShutdownPossible := 	nState <= 10000;
								
IF bCNCMidwareShutdownPossible AND stCNC_Data^.MidwareRequestedShutdown AND (NOT bCNCHandshakeTimeout) THEN
	stCNC_Data^.ApproveShutdownRequest := TRUE;
END_IF

IF stCNC_Data^.ApproveShutdownRequest THEN
	IF bCNCHandshakeTimeout THEN
		bShutdownIsProcessing := TRUE;
	END_IF
END_IF

IF bShutdownIsProcessing THEN
	stCNC_Data^.ApproveShutdownRequest := FALSE;
	stCNC_Data^.MidwareRequestedShutdown := FALSE;
	IF (NOT bCNCHandshakeTimeout) THEN
		bShutdownIsProcessing := FALSE;
	END_IF
END_IF

(*Error handling*)
IF nState > 0 AND nState < 150000 THEN
	nStatePrevious := nState;
END_IF

(*Maintance*)
IF bManualMode THEN
	nState := 150000;
END_IF

(*Emergency*)
IF NOT i_bLO1_Main THEN
	nState := 0;
END_IF

(*Last states*)
IF(nState >= 1000) AND (nState < 150000) THEN
(*Steps before any state*)
	IF anLastStates[0] <> nState THEN
		FOR iLastStates:=500 TO 1 BY -1 DO
			anLastStates[iLastStates]:= anLastStates[iLastStates-1];
		END_FOR
		anLastStates[0]:= nState;
	END_IF
END_IF	

IF fbCncServoVise.bError (*OR stCNC_Data^.ControlStatus_Error*)
THEN
	bError  :=  TRUE;
END_IF



(*   Vise Position Adjustment   *)
fbCncServoVise.nCalOffset_1 := 31.32;	//Originally 22.32
fbCncServoVise.nCalOffset_2 := 108.01;	//Originally 99.01

bCNCRunning := ((nState > 10000) AND (nState <= 30000));

CASE nState OF
{region "Alaphelyzet felvétel"}
	(****************************************************************************************)
	(******************************* Alaphelyzetfelvétel ************************************)
	(****************************************************************************************)	
	0:		(*-----=== Kimenetek törlése ===-----*)
		sState := CONCAT(UDINT_TO_STRING(nState) ,' - A biztonsági kör nem aktív');
		IF i_bLO1_Main AND (NOT bManualMode) THEN		//AND i_bLO1_CNC1 THEN		Nincs bekötve! Teszteléshez kikapcsolva! Ha a bekötés kész VISSZAÍRNI !!!!!!!!!!!!!!!
			stCNC_Data^.DoorControl_CloseDoor := FALSE;
			stCNC_Data^.DoorControl_OpenDoor := FALSE;
			stCNC_Data^.MagazineTable_Trigger := FALSE;
			stCNC_Data^.ToolTable_Trigger := FALSE;
			stCNC_Data^.M401_Acknowledge := FALSE;
			stCNC_Data^.M402_Acknowledge := FALSE;
			stCNC_Data^.M403_Acknowledge := FALSE;
			stCNC_Data^.StartCNCProgram := FALSE;
			stCNC_Data^.StopCNCProgram := FALSE;
			stCNC_Data^.CancelCNCProgram := FALSE;
			stCNC_Data^.SelectCNCProgramByNodeID := FALSE;
			stCNC_Data^.SelectCNCPrograBlockNumber := FALSE;
//			stCNC_Data^.ToolTablePath := '';
			stCNC_Data^.ToolTableLoadTrigger := FALSE;
			stCNC_Data^.MagazineTableLoadTrigger := FALSE;
			stCNC_Data^.ProgramLoadTrigger := FALSE;
			IF bStepEnable THEN
				nState := nState + 20;
			END_IF
		END_IF

	20:		(*-----=== CNC ellenőrzés ===-----*)
		sState := CONCAT(UDINT_TO_STRING(nState) ,' - A CNC ellenőrzése');
		IF stCNC_Data^.ServerState = 'Running' AND
		   stCNC_Data^.CurrentState_State = 'NCIsAvailable' THEN
				IF		stCNC_Data^.CurentState_Program = 'Running' THEN
					nState := 11500;										// A megmunkálás folyamatban -> Várakozás megmunkálás végére.
				ELSIF	stCNC_Data^.CurentState_Program = 'Idle' OR stCNC_Data^.CurentState_Program = 'NotSelected' OR stCNC_Data^.CurentState_Program = 'Interrupted' THEN
					IF (stDutData_Cnc3.nDutId > 0 AND stDutData_Cnc3.bDone) OR stDutData_Cnc3.bDutInVise THEN
						IF bStepEnable THEN									// Késztermék a satuban
							nState := 11560;
						END_IF
					ELSE
						IF bStepEnable THEN									// A satu üres
							nState := nState + 20;
						END_IF
					END_IF
				END_IF
		END_IF

	40:		(*-----=== CNC ajtó nnyitása ===-----*)
		sState := CONCAT(UDINT_TO_STRING(nState) ,' - A CNC ajtó nyitása');
		stCNC_Data^.DoorControl_OpenDoor := TRUE;
		IF stCNC_Data^.DoorControl_DoorOpened THEN
			IF bStepEnable THEN	
				stCNC_Data^.DoorControl_OpenDoor := FALSE;
				nState := nState + 20;
			END_IF
		END_IF

	60:
		nState := 10000;
{endregion}

{region "Alaphelyzet"}
	(****************************************************************************************)
	(*********************************** Alaphelyzet ****************************************)
	(****************************************************************************************)	
	10000:		(*-----=== Várakozás berakásra ===-----*)
		sState := CONCAT(UDINT_TO_STRING(nState) ,' - Várakozás alapanyagra');
		IF ((NOT bShutdownIsProcessing) AND (NOT stCNC_Data^.ApproveShutdownRequest)) THEN
			IF Robot7AxisProgram.bStartCNC3 THEN
				IF stDutData_Cnc3.nDutId > 0 THEN											// Alapanyag a robotnál
					IF bStepEnable THEN	
						nState := 11000;			// -> Alapanyag fogadása
					END_IF
				END_IF
			END_IF
		END_IF
{endregion}

{region "Alapanyag fogadása"}
	(****************************************************************************************)
	(******************************** Alapanyag fogadása ************************************)
	(****************************************************************************************)	
	11000:		(*-----=== Satu pozícionálása ===-----*)
		sState := CONCAT(UDINT_TO_STRING(nState) ,' - Satu pozícionálása');
		fbCncServoVise.nPosition := stDutData_Cnc3.nDimX;
		fbCncServoVise.eCommand := E_CncServoCommand.MovePos;
		IF fbCncServoVise.bDone THEN
			IF bStepEnable THEN
				fbCncServoVise.eCommand := E_CncServoCommand.NoCommand;
				nState := 11100;
			END_IF
		END_IF

	11100:		(*-----=== Várakozás alapanyag berakásra ===-----*)
		sState := CONCAT(UDINT_TO_STRING(nState) ,' - Alapanyag berakás');
		IF Robot7AxisProgram.fbRobot.bZoneCnc3 THEN
			IF bStepEnable THEN
				stDutData_Cnc3.bDutInVise := TRUE;
				nState := 11200;
			END_IF
		END_IF

	11200:		(*-----=== Várakozás robot távozásra ===-----*)
		sState := CONCAT(UDINT_TO_STRING(nState) ,' - Várakozás robot távozásra');
		IF NOT Robot7AxisProgram.fbRobot.bZoneCnc3 THEN
			IF bStepEnable THEN
				nState := 11300;
			END_IF
		END_IF
	
	11300:		(*-----=== Satu rögzítése ===-----*)
		sState := CONCAT(UDINT_TO_STRING(nState) ,' - Satu rögzítése');
		fbCncServoVise.nTorque := stDutData_Cnc3.nTorque;
		fbCncServoVise.eCommand := E_CncServoCommand.Fixed;
		IF fbCncServoVise.bDone THEN
			IF bStepEnable THEN
				fbCncServoVise.eCommand := E_CncServoCommand.NoCommand;
				nState := 11400;
			END_IF
		END_IF

	11400:		(*-----=== CNC ajtó zárása ===-----*)
		sState := CONCAT(UDINT_TO_STRING(nState) ,' - A CNC ajtó zárása');
		stCNC_Data^.DoorControl_CloseDoor := TRUE;
		IF stCNC_Data^.DoorControl_DoorClosed THEN
			IF bStepEnable THEN	
				stCNC_Data^.DoorControl_CloseDoor := FALSE;
				nState := nState + 20;
			END_IF
		END_IF

	11420:		(*-----=== CNC előkészítése ===-----*)
		sState := CONCAT(UDINT_TO_STRING(nState) ,' - A CNC előkészítése');
		IF TRUE THEN															// Külön FB-be rakni mert még képlékeny CAM file letöltése, ellenőrzése, felmásolása, betöltése, ........ 
			IF bStepEnable THEN	
				nState := nState + 20;
			END_IF
		END_IF

	11440:		(*-----=== CAM program indítása ===-----*)
		sState := CONCAT(UDINT_TO_STRING(nState) ,' - CAM program indítása');
		stCNC_Data^.StartCNCProgram := TRUE;
		IF stCNC_Data^.CurentState_Program = 'Running' THEN
			IF bStepEnable THEN	
				stCNC_Data^.StartCNCProgram := FALSE;
				nState := 11500;
			END_IF
		END_IF
	
	11500:		(*-----=== Várakozás CAM program végére ===-----*)
		sState := CONCAT(UDINT_TO_STRING(nState) ,' - Várakozás CAM program végére');
		IF stCNC_Data^.CurentState_Program = 'Finished' OR stCNC_Data^.CurentState_Program = 'Idle' THEN
			IF bStepEnable THEN	
				stCNC_Data^.DoorControl_CloseDoor := FALSE;
				nState := nState + 20;
			END_IF
		END_IF

	11520:		(*-----=== CNC folyamat befejezése ===-----*)
		sState := CONCAT(UDINT_TO_STRING(nState) ,' - A CNC folyamat befejezése');
		IF TRUE THEN															// Külön FB-be rakni mert még képlékeny: minőségellenőrzés, mérési adatok, .... 
			IF bStepEnable THEN	
				nState := nState + 20;
			END_IF
		END_IF

	11540:		(*-----=== CAM program leállítása ===-----*)
		sState := CONCAT(UDINT_TO_STRING(nState) ,' - CAM program leállítása');
		stCNC_Data^.CancelCNCProgram := TRUE;
		IF stCNC_Data^.CurentState_Program = 'Idle' THEN
			IF bStepEnable THEN	
				stCNC_Data^.CancelCNCProgram := FALSE;
				nState := nState + 20;
			END_IF
		END_IF

	11560:		(*-----=== CNC ajtó nnyitása ===-----*)
		sState := CONCAT(UDINT_TO_STRING(nState) ,' - A CNC ajtó nyitása');
		stCNC_Data^.DoorControl_OpenDoor := TRUE;
		IF stCNC_Data^.DoorControl_DoorOpened THEN
			IF bStepEnable THEN	
				stCNC_Data^.DoorControl_OpenDoor := FALSE;
				nState := 11600;
			END_IF
		END_IF
	
	11600:		(*-----=== Satu pozícionálása ===-----*)
		sState := CONCAT(UDINT_TO_STRING(nState) ,' - Satu pozícionálása');
		fbCncServoVise.nPosition := stDutData_Cnc3.nDimX;
		fbCncServoVise.eCommand := E_CncServoCommand.MovePos;
		IF fbCncServoVise.bDone THEN
			IF bStepEnable THEN
				stDutData_Cnc3.bDone := TRUE;
				stDutData_Cnc3.bPass := TRUE;
				fbCncServoVise.eCommand := E_CncServoCommand.NoCommand;
				nState := 12000;
			END_IF
		END_IF
{endregion}

{region "Alapanyag küldése"}
	(****************************************************************************************)
	(******************************** Alapanyag küldése ************************************)
	(****************************************************************************************)	
	12000:		(*-----=== Várakozás alapanyag kivételre ===-----*)
		sState := CONCAT(UDINT_TO_STRING(nState) ,' - Alapanyag kivétel');
		IF Robot7AxisProgram.fbRobot.bZoneCnc3 THEN
			IF bStepEnable THEN
				nState := 12100;
			END_IF
		END_IF
	
	12100:		(*-----=== Várakozás robot távozásra ===-----*)
		sState := CONCAT(UDINT_TO_STRING(nState) ,' - Satu rögzítése');
		IF NOT Robot7AxisProgram.fbRobot.bZoneCnc3 THEN
			IF bStepEnable THEN
				stDutData_Cnc3.bDutInVise := FALSE;
				stDutData_Cnc3.nDutId := 0;
				stDutData_Cnc3.bDone := FALSE;
				nState := 10000;
			END_IF
		END_IF
{endregion}

	150000: (* Maintenance *)
		sState := CONCAT(UDINT_TO_STRING(nState) ,' - Maintenance');
		IF NOT bManualMode THEN
			nState := 0;
		END_IF
		
	200000:(* Error handling *)
		sState := CONCAT(UDINT_TO_STRING(nState) ,CONCAT(' - Error, from this state: ' , sState));
		nState := 200020;

	200020:(* Error handling *)
		IF bAckP THEN
			CASE nStatePrevious OF
				0..9999: nState := 0;
//				10000..25000: nState := 10000;
//				30000..31000: nState := 30000;
			ELSE nState := 0;
			END_CASE
		END_IF	
		
	ELSE //Not a real step, for test purposes
		sState := CONCAT(UDINT_TO_STRING(nState) ,' - Not a real step, for test purposes');
END_CASE

(*Timers***************************************************)
fbCycleTime(IN:= nState > 10000 AND nState <= 95000, PT:= T#1D, Q=> , ET=> );
IF nState > 10000 AND nState <= 95000 THEN
	nCycleTime := TIME_TO_REAL(fbCycleTime.ET)/1000;
END_IF

ServoVise();
//fbCncServoVise.bTestUp := i_bTest_Up;
//fbCncServoVise.bTestDown := i_bTest_Down;
//fbCncServoVise.bTestStop := i_bTest_Stop;

ACTION ServoVise:
fbCncServoVise(
	sName:= 'AWEA_3', 
	bErrorAck:= bAckP, 
	bEnable:= i_bLO1_Main,		//AND i_bLO1_CNC1 THEN		Nincs bekötve! Teszteléshez kikapcsolva! Ha a bekötés kész VISSZAÍRNI !!!!!!!!!!!!!!!, 
	bManualMode:= bManualMode, 
	bReady=> , 
	bBusy=> , 
	bDone=> , 
	bError=> );
END_ACTION

END_PROGRAM

// ---- POUs/RobotKardexStation/RobotKardexProgram.TcPOU
PROGRAM RobotKardexProgram
VAR	(* Control *)
	nState						: UDINT;
	nStatePrevious				: UDINT;
	sState						: STRING(500);
	bError						: BOOL;
	fbCycleTime					: TON;
	nCycleTime					: REAL;
END_VAR
VAR (* Interlock *)
	bInterlock_Strip1			: BOOL;
	bInterlock_Strip2			: BOOL;
	bInterlock_Strip3			: BOOL;
END_VAR
VAR CONSTANT
	iLastStatesMax				: INT := 500;
END_VAR
VAR //LastStates
	anLastStates				:ARRAY[0..iLastStatesMax] OF UDINT;
    iLastStates					:INT;
END_VAR
VAR (* Robot *)
	fbRobot						: FB_Fanuc_Kardex;
	arRobotEvents				: ARRAY [0..15] OF TcEventEntry;
END_VAR
VAR (* Test variables *)
	nOverride					: BYTE := 60;
	nProgNr						: UINT;
	nWeight						: UINT;
	nErrorId					: UDINT;
//	ePath						: E_CNC_Robot_Path;
END_VAR
VAR // MySQL
	
END_VAR

MySQL();

(*Error handling*)
IF nState > 0 AND nState < 150000 THEN
	nStatePrevious := nState;
END_IF

(*Maintance*)
IF bManualMode THEN
	nState := 150000;
END_IF

(*Emergency*)
IF NOT i_bLO1_Main THEN
	nState := 0;
END_IF

(*Last states*)
IF(nState >= 1000) AND (nState < 150000) THEN
(*Steps before any state*)
	IF anLastStates[0] <> nState THEN
		FOR iLastStates:=iLastStatesMax TO 1 BY -1 DO
			anLastStates[iLastStates]:= anLastStates[iLastStates-1];
		END_FOR
		anLastStates[0]:= nState;
	END_IF
END_IF	

IF fbRobot.bError
THEN
	bError  :=  TRUE;
END_IF



CASE nState OF
{region "Alaphelyzet felvétel"}
	(****************************************************************************************)
	(******************************* Alaphelyzetfelvétel ************************************)
	(****************************************************************************************)	
	0:		(*-----=== Kimenetek törlése ===-----*)
		sState := CONCAT(UDINT_TO_STRING(nState) ,' - A biztonsági kör nem aktív');
		bInterlock_Strip1 := TRUE;
		bInterlock_Strip2 := TRUE;
		bInterlock_Strip3 := TRUE;
		IF i_bLO1_Main AND NOT bManualMode AND NOT fbRobot.bPendantMode THEN
			nState := nState + 20;
		END_IF

	20: 
		sState := CONCAT(UDINT_TO_STRING(nState) ,' - Robot alaphelyzetfelvétel');
		fbRobot.eCommand := E_Kardex_Robot_Command.Home;
		IF NOT fbRobot.bBusy AND fbRobot.bReady THEN
			fbRobot.eCommand := E_CNC_Robot_Command.NoCommand;
			bInterlock_Strip1 := FALSE;
			bInterlock_Strip2 := FALSE;
			bInterlock_Strip3 := FALSE;
			nState := nState + 20;
		END_IF
	
	40:
		sState := CONCAT(UDINT_TO_STRING(nState) ,' - Robot megfogó ellenőrzése');
		IF fbRobot.bPartPresent THEN
			nState := 30000;						// Van darab a robotnál -> le kell tenni
		ELSE
			nState := nState + 20;
		END_IF
	
	60:
		nState := 10000;
{endregion}
		
{region "Alaphelyzet"}
	(****************************************************************************************)
	(*********************************** Alaphelyzet ****************************************)
	(****************************************************************************************)	
	10000:		(* -----=== Várakozás parancsra ===----- *)
		sState := CONCAT(UDINT_TO_STRING(nState) ,' - Alaphelyzet');
		IF fbS32.bPalletAtStopper THEN
			bInterlock_Strip1 := TRUE;
			nState := 20000;
		END_IF
{endregion}

{region "bepakolás a CNC-be"}
	(****************************************************************************************)
	(************************** Felső pálya -> Alsó pálya ***********************************)
	(****************************************************************************************)
	20000:		(*-----=== Paletta felvétele felső pályáról ===-----*)
		sState := CONCAT(UDINT_TO_STRING(nState) ,' - Robot felső pálya felvétel');
		fbRobot.nStripNumber := 1;
		fbRobot.eCommand := E_Kardex_Robot_Command.Pick_Up_Strip;
		IF fbRobot.bBusy THEN
			nState := nState + 20;
		END_IF
		
	20020:		(*-----=== Várakozás Robotmozgásra ===-----*)
		sState := CONCAT(UDINT_TO_STRING(nState) ,' - Várakozáas robot mozgásra');
		IF NOT fbRobot.bBusy THEN
			fbRobot.eCommand := E_Kardex_Robot_Command.NoCommand;
			bInterlock_Strip3 := TRUE;
			nState := 30000;
		END_IF
	
	30000:		(*-----=== Várakozás lerakási engedélyre ===-----*)
		sState := CONCAT(UDINT_TO_STRING(nState) ,' - Várakozáas robot mozgásra');
		IF NOT fbS23.i_bPalettSensor AND NOT fbs22.bPalletSent THEN
			nState := nState + 20;
		END_IF
	
	30020:
		bInterlock_Strip1 := FALSE;
		nState := 40000;
	
	40000:		(*-----=== Paletta lerakása alsó pályára ===-----*)
		sState := CONCAT(UDINT_TO_STRING(nState) ,' - Robot alsó pálya lerakás');
		fbRobot.nStripNumber := 3;
		fbRobot.eCommand := E_Kardex_Robot_Command.Put_Down_Strip;
		IF fbRobot.bBusy THEN
			nState := nState + 20;
		END_IF
		
	40020:		(*-----=== Várakozás Robotmozgásra ===-----*)
		sState := CONCAT(UDINT_TO_STRING(nState) ,' - Várakozáas robot mozgásra');
		IF NOT fbRobot.bBusy THEN
			fbRobot.eCommand := E_Kardex_Robot_Command.NoCommand;
			bInterlock_Strip3 := FALSE;
			nState := 50000;
		END_IF
	
	50000:
		nState := 10000;
	
	150000: (* Maintenance *)
		sState := CONCAT(UDINT_TO_STRING(nState) ,' - Maintenance');
		IF NOT bManualMode THEN
			nState := 0;
		END_IF
		
	200000:(* Error handling *)
		sState := CONCAT(UDINT_TO_STRING(nState) ,CONCAT(' - Error, from this state: ' , sState));
		nState := 200020;
	
	200020:(* Error handling *)
		IF bAckP THEN
			CASE nStatePrevious OF
				0..9999: nState := 0;
//				10000..25000: nState := 10000;
//				30000..31000: nState := 30000;
			ELSE nState := 0;
			END_CASE
		END_IF	
		
	ELSE //Not a real step, for test purposes
		sState := CONCAT(UDINT_TO_STRING(nState) ,' - Not a real step, for test purposes');
END_CASE

(*Timers***************************************************)
fbCycleTime(IN:= nState > 10000 AND nState <= 95000, PT:= T#1D, Q=> , ET=> );
IF nState > 10000 AND nState <= 95000 THEN
	nCycleTime := TIME_TO_REAL(fbCycleTime.ET)/1000;
END_IF

Robot();

ACTION MySQL:
;
END_ACTION

ACTION Robot:
arRobotEvents[0] := TC_EVENTS.MyEvents.RobotNoPneumaticsErr;
arRobotEvents[1] := TC_EVENTS.MyEvents.RobotNotCorrectPrgErr;
arRobotEvents[2] := TC_EVENTS.MyEvents.RobotNotProdOnRobotErr;
arRobotEvents[3] := TC_EVENTS.MyEvents.RobotProdOnRobotErr;
arRobotEvents[4] := TC_EVENTS.MyEvents.RobotGripperOpenErr;
arRobotEvents[5] := TC_EVENTS.MyEvents.RobotGripperCloseErr;
arRobotEvents[6] := TC_EVENTS.MyEvents.RobotNotCorrectViseNumberErr;
arRobotEvents[7] := TC_EVENTS.MyEvents.RobotNotReadyErr;
arRobotEvents[8] := TC_EVENTS.MyEvents.RobotBasePosErr;


(*-----=== Hand shake jelek kezelése ===-----*)
fbRobot.bKardex_Reset := fbRobot.bKardex_Set;							// 05.1	Robot Kardex-be menne
fbRobot.bHolder_Reset := fbRobot.bHolder_Set;							// 05.1	Robot Kardex-be menne
fbRobot.bMir_Reset := fbRobot.bMir_Set;									// 05.1	Robot Kardex-be menne
fbRobot.bStrip_1_Reset := fbRobot.bStrip_1_Set;							// 05.1	Robot Kardex-be menne
fbRobot.bStrip_2_Reset := fbRobot.bStrip_2_Set;							// 05.1	Robot Kardex-be menne
fbRobot.bStrip_3_Reset := fbRobot.bStrip_3_Set;							// 05.1	Robot Kardex-be menne


fbRobot(
	sName:= 'Fanuc - Kardex', 
	bEn:= i_bLO2_Main, 
	timeBaseState:= T#40S, 
	bAck:= bAckP, 
	bOverride:= nOverride, 
	stEventArray:= arRobotEvents);
END_ACTION

END_PROGRAM

// ---- POUs/FBs/FanucKardex/FB_Fanuc_Kardex.TcPOU
FUNCTION_BLOCK FB_Fanuc_Kardex
VAR_INPUT
	sName				:STRING;
	bEn					:BOOL;				(* Engedély jel *)
	eCommand			:E_Kardex_Robot_Command;	(* Végrehajtandó parancsok *)	
	nKardexFloor		:BYTE;				(* Kardex tálca sorszáma (1-50) *)
	nKardexJigNumber	:BYTE;				(* Kardex ülék sorszáma (1-30) *)
	nMirNumber			:BYTE;				(* MIR száma; 1 vagy 2 *)
	nMir_JigNumber		:BYTE;				(* Mir paletta szám (1-4) *)
	nPufferNumber		:BYTE;				(* Puffer tároló paletta szám (1-15) *)
	nStripNumber		:BYTE;				(* Szalag száma (1-3) *)
	bKardex_Reset		:BOOL;				(* Handshake *)
	bMir_1_Reset		:BOOL;				(* Handshake *)
	bMir_2_Reset		:BOOL;				(* Handshake *)
	bPuffer_Reset		:BOOL;				(* Handshake *)
	bStrip_1_Reset		:BOOL;				(* Handshake *)
	bStrip_2_Reset		:BOOL;				(* Handshake *)
	bStrip_3_Reset		:BOOL;				(* Handshake *)	
	timeBaseState		:TIME:=T#20S;		(* Alaphelyzet felvételi idő*)
	bAck				:BOOL; 				(* Hibanyugta *)
	bOverride			:BYTE := 10;		(* PLC Override  10 - 100%*)
	stEventArray		:ARRAY [0..nMaxAlarmNr] OF TcEventEntry;	(* Event array definition *)
END_VAR
VAR_OUTPUT
	bReady				:BOOL;				(* Folyamat üzemkész *)
	bBusy				:BOOL;				(* Folyamat aktív *)
	bDone				:BOOL;				(* Folyamat kész *)
	bPendantMode		:BOOL;				(* Teach pendant mód aktív *)
	bKardex_Set			:BIT;				(* Handshake *)
	bMir_1_Set			:BIT;				(* Handshake *)
	bMir_2_Set			:BIT;				(* Handshake *)
	bPuffer_Set			:BIT;				(* Handshake *)
	bStrip_1_Set		:BIT;				(* Handshake *)
	bStrip_2_Set		:BIT;				(* Handshake *)
	bStrip_3_Set		:BIT;				(* Handshake *)
	bError				:BOOL;				(* Hiba bit*)
	sError				:STRING(255);		(* Hiba string*)
END_VAR
VAR CONSTANT
	nMaxAlarmNr			:INT := 15;
END_VAR
VAR (* Robot IO *)
	RobotIn				:U_Kardex_Fanuc_Input;
	RobotOut			:U_Kardex_Fanuc_Output;
END_VAR
VAR (* State control *)
	tBaseState			:TON;
	tResetFault			:TON;
	tStopCycle			:TON;
	tStartCycle			:TON;
	
	nState				:UDINT;
	sState				:STRING;
	bIsInitalized		:BOOL;
	bRobotReady			:BOOL;
END_VAR
VAR (* Error handling*)
	bErrNotReady		:BOOL;
	bErrBaseTimeout		:BOOL;
	fbAlarmArray		:ARRAY [0..nMaxAlarmNr] OF FB_TcAlarm;
	arrAlarms			:ARRAY [0..nMaxAlarmNr] OF BOOL;
	i					:INT;
	
	//LastStates
	anLastStates				:ARRAY[0..500] OF UDINT;
    iLastStates					:INT;
END_VAR

(*Handshake**************************************************)
bKardex_Set := RobotIn.Status.bKardex_Set;
bMir_1_Set := RobotIn.Status.bMir_1_Set;
bMir_2_Set := RobotIn.Status.bMir_2_Set;
bPuffer_Set := RobotIn.Status.bPuffer_Set;
bStrip_1_Set := RobotIn.Status.bStrip_1_Set;
bStrip_2_Set := RobotIn.Status.bStrip_2_Set;
bStrip_3_Set := RobotIn.Status.bStrip_3_Set;
RobotOut.Control.bKardex_Reset := bKardex_Reset;
RobotOut.Control.bMir_1_Reset := bMir_1_Reset;
RobotOut.Control.bMir_2_Reset := bMir_2_Reset;
RobotOut.Control.bPuffer_Reset := bPuffer_Reset;
RobotOut.Control.bStrip_1_Reset := bStrip_1_Reset;
RobotOut.Control.bStrip_2_Reset := bStrip_2_Reset;
RobotOut.Control.bStrip_3_Reset := bStrip_3_Reset;

(*Időzítők***************************************************)
tBaseState(IN:= (nState > 0 AND nState < 10000), PT:= timeBaseState);
tResetFault(IN:= RobotOut.Control.bReset, PT:= T#100MS);
tStopCycle(IN:= RobotOut.Control.bCycleStop, PT:= T#100MS);
tStartCycle(IN:= RobotOut.Control.bStart, PT:= T#100MS);

(*Vész rendszer**************************************************)
bRobotReady :=  NOT RobotIn.Status.bControllerEmyStop AND
				NOT RobotIn.Status.bTeachPendantEmyStop AND
				NOT RobotIn.Status.bDeadman AND
				NOT RobotIn.Status.bFence AND
				NOT RobotIn.Status.bEmyStopExternal;
				
(*Hibakezelés************************************************)
IF nState >= 200 AND nState < 150000 AND (RobotIn.Status.bAlarm OR RobotIn.Status.bFault OR NOT bRobotReady) THEN
	bErrNotReady := TRUE;
END_IF

IF tBaseState.Q AND NOT bErrBaseTimeout THEN
	bErrBaseTimeout := TRUE;
END_IF

bError := (RobotIn.Status.bAlarm AND bEn) OR
			RobotIn.Status.bNoPneumatics OR
			RobotIn.Status.bNotCorrectPrg OR
			RobotIn.Status.bNotProductOnRobot OR
			RobotIn.Status.bProductOnRobot OR
			RobotIn.Status.bGripperOpenError OR
			RobotIn.Status.bGripperCloseError OR
			RobotIn.Status.bPartPresentError OR
			RobotIn.Status.bNotCorrectKardexFloor OR
			RobotIn.Status.bNotCorrectKardexJig OR
			RobotIn.Status.bNotCorrectMir OR
			RobotIn.Status.bNotCorrectPuffer OR
			bErrNotReady OR
			bErrBaseTimeout;

arrAlarms[0] := RobotIn.Status.bNoPneumatics;			
arrAlarms[1] := RobotIn.Status.bNotCorrectPrg;
arrAlarms[2] := RobotIn.Status.bNotProductOnRobot;
arrAlarms[3] := RobotIn.Status.bProductOnRobot;
arrAlarms[4] := RobotIn.Status.bGripperOpenError;
arrAlarms[5] := RobotIn.Status.bGripperCloseError;
arrAlarms[6] := RobotIn.Status.bPartPresentError;
arrAlarms[7] := RobotIn.Status.bNotCorrectKardexFloor;
arrAlarms[8] := RobotIn.Status.bNotCorrectKardexJig;
arrAlarms[9] := RobotIn.Status.bNotCorrectMir;
arrAlarms[10] := RobotIn.Status.bNotCorrectPuffer;
arrAlarms[11] := bErrNotReady;
arrAlarms[12] := bErrBaseTimeout;

IF nState > 140 AND nState < 150000 AND bError THEN
	nState := 200000;
END_IF
					
(*State history ************************************************)
IF(nState >= 100) AND (nState <= 20000) THEN
(*Steps before any state*)
	IF anLastStates[0] <> nState THEN
		FOR iLastStates:=500 TO 1 BY -1 DO
			anLastStates[iLastStates]:= anLastStates[iLastStates-1];
		END_FOR
		anLastStates[0]:= nState;
	END_IF
END_IF	

(*Pendant mód ************************************************)
bPendantMode := RobotIn.Status.bPendant;
IF bPendantMode THEN
	nState := 150000;
END_IF

(*Engedélyek *************************************************)
IF (NOT bEn AND NOT bPendantMode) THEN			// nincs ajtókör, és pendantról sem szeretnék használni
	nState := 0;
END_IF

// Enable signals
RobotOut.Control.bZoneEnable := bEn;
RobotOut.Control.bPlcOverride := bOverride;

(*Automata üzem *********************************************)
CASE nState OF
	(* Emergency circuit broken - Base state *)
	0:(* Operation stop - Emergency circuit check *)
		sState := CONCAT(UDINT_TO_STRING(nState) ,' - Vészkör vagy ajtókör bontva - Működtetések törlése');
		RobotOut.Control.bImmediateStop := FALSE;
		RobotOut.Control.bHold := FALSE;
		RobotOut.Control.bSafeSpeed := FALSE;
		RobotOut.Control.bCycleStop := FALSE;
		RobotOut.Control.bReset := FALSE;
		RobotOut.Control.bStart := FALSE;
		RobotOut.Control.bPNS1 := TRUE;
		RobotOut.Control.bPNS2 := FALSE;
		RobotOut.Control.bPNS3 := FALSE;
		RobotOut.Control.bPNS4 := FALSE;
		RobotOut.Control.bPNS5 := FALSE;
		RobotOut.Control.bPNS6 := FALSE;
		RobotOut.Control.bPNS7 := FALSE;
		RobotOut.Control.bPNS8 := FALSE;
		RobotOut.Control.bPnsStrobe := FALSE;
		RobotOut.Control.bEnable := FALSE;
		RobotOut.Control.bHome := FALSE;
		RobotOut.Control.bServiceEnd := FALSE;
		RobotOut.Control.nMode := 0;
		RobotOut.Control.nProgramNumber := 0;
		RobotOut.Control.bProdStart := FALSE;
		RobotOut.Control.bKardex_Reset := FALSE;
		RobotOut.Control.bMir_1_Reset := FALSE;
		RobotOut.Control.bMir_2_Reset := FALSE;
		RobotOut.Control.bPuffer_Reset := FALSE;
		RobotOut.Control.bStrip_1_Reset := FALSE;
		RobotOut.Control.bStrip_2_Reset := FALSE;
		RobotOut.Control.bStrip_3_Reset := FALSE;
		bErrNotReady := FALSE;
		bErrBaseTimeout := FALSE;
		bReady := FALSE;
		bBusy := FALSE;	
		IF bEn AND bRobotReady THEN
			bBusy := TRUE;
			nState := nState + 20;
		END_IF
		
